LIN {X 0,Y 563.964,Z 599.477,A -85,B 0,C 180,E1 22437.391,E2 22437.391} C_VEL
LIN {X 0,Y 563.324,Z 620.016,A -85,B 0,C 180,E1 22436.115,E2 22436.115} C_VEL
LIN {X 0,Y 562.702,Z 638.754,A -85,B 0,C 180,E1 22434.736,E2 22434.736} C_VEL
LIN {X 0,Y 562.109,Z 656.522,A -85,B 0,C 180,E1 22433.203,E2 22433.203} C_VEL
LIN {X 0,Y 561.587,Z 672.775,A -85,B 0,C 180,E1 22431.57,E2 22431.57} C_VEL
LIN {X 0,Y 561.094,Z 689.022,A -85,B 0,C 180,E1 22429.681,E2 22429.681} C_VEL
LIN {X 0,Y 560.721,Z 703.041,A -85,B 0,C 180,E1 22427.784,E2 22427.784} C_VEL
LIN {X 0,Y 560.419,Z 715.335,A -85,B 0,C 180,E1 22425.841,E2 22425.841} C_VEL
LIN {X 0,Y 560.206,Z 726.094,A -85,B 0,C 180,E1 22423.837,E2 22423.837} C_VEL
LIN {X 0,Y 560.064,Z 735.578,A -85,B 0,C 180,E1 22421.742,E2 22421.742} C_VEL
LIN {X 0,Y 559.974,Z 743.231,A -85,B 0,C 180,E1 22419.662,E2 22419.662} C_VEL
LIN {X 0,Y 559.926,Z 749.535,A -85,B 0,C 180,E1 22417.49,E2 22417.49} C_VEL
LIN {X 0,Y 559.914,Z 754.246,A -85,B 0,C 180,E1 22415.328,E2 22415.328} C_VEL
LIN {X 0,Y 559.914,Z 757.235,A -85,B 0,C 180,E1 22413.173,E2 22413.173} C_VEL
LIN {X 0,Y 559.911,Z 758.795,A -85,B 0,C 180,E1 22410.921,E2 22410.921} C_VEL
LIN {X 0,Y 559.913,Z 758.748,A -85,B 0,C 180,E1 22408.772,E2 22408.772} C_VEL
LIN {X 0,Y 559.916,Z 757.071,A -85,B 0,C 180,E1 22406.586,E2 22406.586} C_VEL
LIN {X 0,Y 559.922,Z 753.812,A -85,B 0,C 180,E1 22404.364,E2 22404.364} C_VEL
LIN {X 0,Y 559.93,Z 749.248,A -85,B 0,C 180,E1 22402.304,E2 22402.304} C_VEL
LIN {X 0,Y 559.978,Z 742.83,A -85,B 0,C 180,E1 22400.13,E2 22400.13} C_VEL
LIN {X 0,Y 560.079,Z 735.084,A -85,B 0,C 180,E1 22398.041,E2 22398.041} C_VEL
LIN {X 0,Y 560.224,Z 725.498,A -85,B 0,C 180,E1 22395.953,E2 22395.953} C_VEL
LIN {X 0,Y 560.45,Z 713.965,A -85,B 0,C 180,E1 22393.841,E2 22393.841} C_VEL
LIN {X 0,Y 560.763,Z 701.306,A -85,B 0,C 180,E1 22391.871,E2 22391.871} C_VEL
LIN {X 0,Y 561.156,Z 687.174,A -85,B 0,C 180,E1 22389.996,E2 22389.996} C_VEL
LIN {X 0,Y 561.628,Z 671.445,A -85,B 0,C 180,E1 22388.197,E2 22388.197} C_VEL
LIN {X 0,Y 562.193,Z 653.882,A -85,B 0,C 180,E1 22386.468,E2 22386.468} C_VEL
LIN {X 0,Y 562.78,Z 636.185,A -85,B 0,C 180,E1 22384.97,E2 22384.97} C_VEL
LIN {X 0,Y 563.41,Z 617.535,A -85,B 0,C 180,E1 22383.626,E2 22383.626} C_VEL
LIN {X 0,Y 564.028,Z 597.68,A -85,B 0,C 180,E1 22382.419,E2 22382.419} C_VEL
LIN {X 0,Y 564.627,Z 577.104,A -85,B 0,C 180,E1 22381.38,E2 22381.38} C_VEL
LIN {X 0,Y 565.175,Z 556.456,A -85,B 0,C 180,E1 22380.541,E2 22380.541} C_VEL
LIN {X 0,Y 565.571,Z 535.019,A -85,B 0,C 180,E1 22379.871,E2 22379.871} C_VEL
LIN {X 0,Y 565.962,Z 512.641,A -85,B 0,C 180,E1 22379.375,E2 22379.375} C_VEL
LIN {X 0,Y 567.326,Z 287.147,A -85,B 0,C 180,E1 22376.127,E2 22376.127} C_VEL
LIN {X 0,Y 567.586,Z 216.731,A -85,B 0,C 180,E1 22375.087,E2 22375.087} C_VEL
LIN {X 0,Y 566.157,Z 208.127,A -85,B 0,C 180,E1 22374.819,E2 22374.819} C_VEL
LIN {X 0,Y 567.277,Z 159.958,A -85,B 0,C 180,E1 22371.59,E2 22371.59} C_VEL
LIN {X 0,Y 567.466,Z 148.971,A -85,B 0,C 180,E1 22370.829,E2 22370.829} C_VEL
LIN {X 0,Y 560.322,Z 132.731,A -85,B 0,C 180,E1 22369.009,E2 22369.009} C_VEL
LIN {X 0,Y 560.266,Z 132.249,A -85,B 0,C 180,E1 22368.542,E2 22368.542} C_VEL
LIN {X 0,Y 560.213,Z 132.266,A -85,B 0,C 180,E1 22365.408,E2 22365.408} C_VEL
LIN {X 0,Y 560.208,Z 132.264,A -85,B 0,C 180,E1 22362.013,E2 22362.013} C_VEL
LIN {X 0,Y 560.234,Z 132.255,A -85,B 0,C 180,E1 22359.051,E2 22359.051} C_VEL
LIN {X 0,Y 560.198,Z 132.249,A -85,B 0,C 180,E1 22355.833,E2 22355.833} C_VEL
LIN {X 0,Y 560.268,Z 132.256,A -85,B 0,C 180,E1 22352.612,E2 22352.612} C_VEL
LIN {X 0,Y 560.213,Z 132.257,A -85,B 0,C 180,E1 22349.431,E2 22349.431} C_VEL
LIN {X 0,Y 560.218,Z 132.25,A -85,B 0,C 180,E1 22346.044,E2 22346.044} C_VEL
LIN {X 0,Y 560.268,Z 132.259,A -85,B 0,C 180,E1 22342.895,E2 22342.895} C_VEL
LIN {X 0,Y 560.215,Z 132.25,A -85,B 0,C 180,E1 22339.714,E2 22339.714} C_VEL
LIN {X 0,Y 560.268,Z 132.258,A -85,B 0,C 180,E1 22336.484,E2 22336.484} C_VEL
LIN {X 0,Y 560.235,Z 132.258,A -85,B 0,C 180,E1 22333.311,E2 22333.311} C_VEL
LIN {X 0,Y 560.23,Z 132.257,A -85,B 0,C 180,E1 22329.969,E2 22329.969} C_VEL
LIN {X 0,Y 560.286,Z 132.258,A -85,B 0,C 180,E1 22326.764,E2 22326.764} C_VEL
LIN {X 0,Y 560.235,Z 132.256,A -85,B 0,C 180,E1 22323.479,E2 22323.479} C_VEL
LIN {X 0,Y 560.244,Z 132.253,A -85,B 0,C 180,E1 22320.102,E2 22320.102} C_VEL
LIN {X 0,Y 560.282,Z 132.256,A -85,B 0,C 180,E1 22316.829,E2 22316.829} C_VEL
LIN {X 0,Y 560.241,Z 132.258,A -85,B 0,C 180,E1 22313.544,E2 22313.544} C_VEL
LIN {X 0,Y 560.263,Z 132.251,A -85,B 0,C 180,E1 22310.239,E2 22310.239} C_VEL
LIN {X 0,Y 560.279,Z 132.254,A -85,B 0,C 180,E1 22306.901,E2 22306.901} C_VEL
LIN {X 0,Y 560.246,Z 132.247,A -85,B 0,C 180,E1 22303.622,E2 22303.622} C_VEL
LIN {X 0,Y 560.274,Z 132.25,A -85,B 0,C 180,E1 22300.288,E2 22300.288} C_VEL
LIN {X 0,Y 560.28,Z 132.252,A -85,B 0,C 180,E1 22296.995,E2 22296.995} C_VEL
LIN {X 0,Y 560.254,Z 132.254,A -85,B 0,C 180,E1 22293.731,E2 22293.731} C_VEL
LIN {X 0,Y 560.283,Z 132.253,A -85,B 0,C 180,E1 22290.375,E2 22290.375} C_VEL
LIN {X 0,Y 560.278,Z 132.249,A -85,B 0,C 180,E1 22287.006,E2 22287.006} C_VEL
LIN {X 0,Y 560.26,Z 132.252,A -85,B 0,C 180,E1 22283.666,E2 22283.666} C_VEL
LIN {X 0,Y 560.28,Z 132.251,A -85,B 0,C 180,E1 22280.292,E2 22280.292} C_VEL
LIN {X 0,Y 560.268,Z 132.254,A -85,B 0,C 180,E1 22276.882,E2 22276.882} C_VEL
LIN {X 0,Y 560.269,Z 132.252,A -85,B 0,C 180,E1 22273.538,E2 22273.538} C_VEL
LIN {X 0,Y 560.346,Z 132.693,A -85,B 0,C 180,E1 22273.213,E2 22273.213} C_VEL
LIN {X 0,Y 561.705,Z 135.907,A -85,B 0,C 180,E1 22272.83,E2 22272.83} C_VEL
LIN {X 0,Y 568.634,Z 150.292,A -85,B 0,C 180,E1 22271.207,E2 22271.207} C_VEL
LIN {X 0,Y 568.491,Z 162.115,A -85,B 0,C 180,E1 22270.464,E2 22270.464} C_VEL
LIN {X 0,Y 570.272,Z 172.641,A -85,B 0,C 180,E1 22270.141,E2 22270.141} C_VEL
LIN {X 0,Y 568.756,Z 379.763,A -85,B 0,C 180,E1 22266.99,E2 22266.99} C_VEL
LIN {X 0,Y 567.81,Z 510.946,A -85,B 0,C 180,E1 22265.019,E2 22265.019} C_VEL
LIN {X 0,Y 567.322,Z 534.795,A -85,B 0,C 180,E1 22264.471,E2 22264.471} C_VEL
LIN {X 0,Y 566.849,Z 556.769,A -85,B 0,C 180,E1 22263.779,E2 22263.779} C_VEL
LIN {X 0,Y 566.165,Z 578.711,A -85,B 0,C 180,E1 22262.891,E2 22262.891} C_VEL
LIN {X 0,Y 565.506,Z 599.807,A -85,B 0,C 180,E1 22261.854,E2 22261.854} C_VEL
LIN {X 0,Y 564.723,Z 620.862,A -85,B 0,C 180,E1 22260.604,E2 22260.604} C_VEL
LIN {X 0,Y 563.958,Z 641.417,A -85,B 0,C 180,E1 22259.179,E2 22259.179} C_VEL
LIN {X 0,Y 563.248,Z 659.599,A -85,B 0,C 180,E1 22257.715,E2 22257.715} C_VEL
LIN {X 0,Y 562.523,Z 678.969,A -85,B 0,C 180,E1 22255.922,E2 22255.922} C_VEL
LIN {X 0,Y 561.905,Z 696.173,A -85,B 0,C 180,E1 22254.1,E2 22254.1} C_VEL
LIN {X 0,Y 561.361,Z 712.099,A -85,B 0,C 180,E1 22252.152,E2 22252.152} C_VEL
LIN {X 0,Y 560.903,Z 727.34,A -85,B 0,C 180,E1 22250.014,E2 22250.014} C_VEL
LIN {X 0,Y 560.562,Z 740.01,A -85,B 0,C 180,E1 22247.973,E2 22247.973} C_VEL
LIN {X 0,Y 560.301,Z 751.321,A -85,B 0,C 180,E1 22245.844,E2 22245.844} C_VEL
LIN {X 0,Y 560.136,Z 761.456,A -85,B 0,C 180,E1 22243.628,E2 22243.628} C_VEL
LIN {X 0,Y 560.026,Z 769.7,A -85,B 0,C 180,E1 22241.429,E2 22241.429} C_VEL
LIN {X 0,Y 559.964,Z 776.775,A -85,B 0,C 180,E1 22239.144,E2 22239.144} C_VEL
LIN {X 0,Y 559.928,Z 782.07,A -85,B 0,C 180,E1 22236.86,E2 22236.86} C_VEL
LIN {X 0,Y 559.899,Z 785.913,A -85,B 0,C 180,E1 22234.609,E2 22234.609} C_VEL
LIN {X 0,Y 559.904,Z 788.122,A -85,B 0,C 180,E1 22232.354,E2 22232.354} C_VEL
LIN {X 0,Y 559.91,Z 788.984,A -85,B 0,C 180,E1 22230.102,E2 22230.102} C_VEL
LIN {X 0,Y 559.905,Z 788.189,A -85,B 0,C 180,E1 22227.749,E2 22227.749} C_VEL
LIN {X 0,Y 559.898,Z 786.049,A -85,B 0,C 180,E1 22225.493,E2 22225.493} C_VEL
LIN {X 0,Y 559.927,Z 782.254,A -85,B 0,C 180,E1 22223.232,E2 22223.232} C_VEL
LIN {X 0,Y 559.952,Z 777.296,A -85,B 0,C 180,E1 22221.063,E2 22221.063} C_VEL
LIN {X 0,Y 560.019,Z 770.409,A -85,B 0,C 180,E1 22218.778,E2 22218.778} C_VEL
LIN {X 0,Y 560.125,Z 762.439,A -85,B 0,C 180,E1 22216.62,E2 22216.62} C_VEL
LIN {X 0,Y 560.282,Z 752.364,A -85,B 0,C 180,E1 22214.368,E2 22214.368} C_VEL
LIN {X 0,Y 560.548,Z 741.242,A -85,B 0,C 180,E1 22212.241,E2 22212.241} C_VEL
LIN {X 0,Y 560.885,Z 728.049,A -85,B 0,C 180,E1 22210.094,E2 22210.094} C_VEL
LIN {X 0,Y 561.317,Z 713.542,A -85,B 0,C 180,E1 22208.034,E2 22208.034} C_VEL
LIN {X 0,Y 561.815,Z 698.473,A -85,B 0,C 180,E1 22206.172,E2 22206.172} C_VEL
LIN {X 0,Y 562.437,Z 681.124,A -85,B 0,C 180,E1 22204.294,E2 22204.294} C_VEL
LIN {X 0,Y 563.12,Z 663.258,A -85,B 0,C 180,E1 22202.596,E2 22202.596} C_VEL
LIN {X 0,Y 563.845,Z 644.352,A -85,B 0,C 180,E1 22201.047,E2 22201.047} C_VEL
LIN {X 0,Y 564.609,Z 623.62,A -85,B 0,C 180,E1 22199.572,E2 22199.572} C_VEL
LIN {X 0,Y 565.353,Z 603.85,A -85,B 0,C 180,E1 22198.375,E2 22198.375} C_VEL
LIN {X 0,Y 566.073,Z 581.179,A -85,B 0,C 180,E1 22197.22,E2 22197.22} C_VEL
LIN {X 0,Y 566.763,Z 559.797,A -85,B 0,C 180,E1 22196.333,E2 22196.333} C_VEL
LIN {X 0,Y 567.282,Z 536.967,A -85,B 0,C 180,E1 22195.59,E2 22195.59} C_VEL
LIN {X 0,Y 567.779,Z 514.194,A -85,B 0,C 180,E1 22195.039,E2 22195.039} C_VEL
LIN {X 0,Y 568.146,Z 469.081,A -85,B 0,C 180,E1 22194.337,E2 22194.337} C_VEL
LIN {X 0,Y 569.615,Z 259.273,A -85,B 0,C 180,E1 22191.19,E2 22191.19} C_VEL
LIN {X 0,Y 570.101,Z 170.611,A -85,B 0,C 180,E1 22189.812,E2 22189.812} C_VEL
LIN {X 0,Y 568.377,Z 161.3,A -85,B 0,C 180,E1 22189.504,E2 22189.504} C_VEL
LIN {X 0,Y 568.463,Z 149.871,A -85,B 0,C 180,E1 22188.749,E2 22188.749} C_VEL
LIN {X 0,Y 561.602,Z 135.762,A -85,B 0,C 180,E1 22187.15,E2 22187.15} C_VEL
LIN {X 0,Y 560.314,Z 132.511,A -85,B 0,C 180,E1 22186.748,E2 22186.748} C_VEL
LIN {X 0,Y 560.271,Z 132.249,A -85,B 0,C 180,E1 22183.539,E2 22183.539} C_VEL
LIN {X 0,Y 560.263,Z 132.252,A -85,B 0,C 180,E1 22180.2,E2 22180.2} C_VEL
LIN {X 0,Y 560.278,Z 132.247,A -85,B 0,C 180,E1 22176.842,E2 22176.842} C_VEL
LIN {X 0,Y 560.275,Z 132.254,A -85,B 0,C 180,E1 22173.465,E2 22173.465} C_VEL
LIN {X 0,Y 560.258,Z 132.257,A -85,B 0,C 180,E1 22170.216,E2 22170.216} C_VEL
LIN {X 0,Y 560.276,Z 132.246,A -85,B 0,C 180,E1 22166.954,E2 22166.954} C_VEL
LIN {X 0,Y 560.282,Z 132.253,A -85,B 0,C 180,E1 22163.562,E2 22163.562} C_VEL
LIN {X 0,Y 560.25,Z 132.254,A -85,B 0,C 180,E1 22160.256,E2 22160.256} C_VEL
LIN {X 0,Y 560.276,Z 132.252,A -85,B 0,C 180,E1 22156.911,E2 22156.911} C_VEL
LIN {X 0,Y 560.283,Z 132.247,A -85,B 0,C 180,E1 22153.519,E2 22153.519} C_VEL
LIN {X 0,Y 560.245,Z 132.254,A -85,B 0,C 180,E1 22150.176,E2 22150.176} C_VEL
LIN {X 0,Y 560.274,Z 132.257,A -85,B 0,C 180,E1 22146.867,E2 22146.867} C_VEL
LIN {X 0,Y 560.278,Z 132.253,A -85,B 0,C 180,E1 22143.478,E2 22143.478} C_VEL
LIN {X 0,Y 560.236,Z 132.255,A -85,B 0,C 180,E1 22140.204,E2 22140.204} C_VEL
LIN {X 0,Y 560.271,Z 132.257,A -85,B 0,C 180,E1 22136.931,E2 22136.931} C_VEL
LIN {X 0,Y 560.263,Z 132.256,A -85,B 0,C 180,E1 22133.647,E2 22133.647} C_VEL
LIN {X 0,Y 560.229,Z 132.258,A -85,B 0,C 180,E1 22130.342,E2 22130.342} C_VEL
LIN {X 0,Y 560.283,Z 132.26,A -85,B 0,C 180,E1 22127.11,E2 22127.11} C_VEL
LIN {X 0,Y 560.232,Z 132.258,A -85,B 0,C 180,E1 22123.941,E2 22123.941} C_VEL
LIN {X 0,Y 560.224,Z 132.25,A -85,B 0,C 180,E1 22120.503,E2 22120.503} C_VEL
LIN {X 0,Y 560.287,Z 132.258,A -85,B 0,C 180,E1 22117.307,E2 22117.307} C_VEL
LIN {X 0,Y 560.217,Z 132.257,A -85,B 0,C 180,E1 22116.289,E2 22116.289} C_VEL
LIN {X 0,Y 559.235,Z 132.381,A -85,B 0,C 180,E1 22115.501,E2 22115.501} C_VEL
LIN {X 0,Y 552.763,Z 133.196,A -85,B 0,C 180,E1 22113.232,E2 22113.232} C_VEL
LIN {X 0,Y 552.295,Z 133.251,A -85,B 0,C 180,E1 22112.713,E2 22112.713} C_VEL
LIN {X 0,Y 552.301,Z 133.241,A -85,B 0,C 180,E1 22109.663,E2 22109.663} C_VEL
LIN {X 0,Y 552.271,Z 133.251,A -85,B 0,C 180,E1 22106.358,E2 22106.358} C_VEL
LIN {X 0,Y 552.33,Z 133.239,A -85,B 0,C 180,E1 22103.141,E2 22103.141} C_VEL
LIN {X 0,Y 552.268,Z 133.241,A -85,B 0,C 180,E1 22099.978,E2 22099.978} C_VEL
LIN {X 0,Y 552.265,Z 133.242,A -85,B 0,C 180,E1 22096.53,E2 22096.53} C_VEL
LIN {X 0,Y 552.324,Z 133.233,A -85,B 0,C 180,E1 22093.303,E2 22093.303} C_VEL
LIN {X 0,Y 552.333,Z 133.515,A -85,B 0,C 180,E1 22091.614,E2 22091.614} C_VEL
LIN {X 0,Y 553.79,Z 136.97,A -85,B 0,C 180,E1 22091.159,E2 22091.159} C_VEL
LIN {X 0,Y 560.859,Z 152.929,A -85,B 0,C 180,E1 22089.346,E2 22089.346} C_VEL
LIN {X 0,Y 559.535,Z 198.989,A -85,B 0,C 180,E1 22086.197,E2 22086.197} C_VEL
LIN {X 0,Y 559.443,Z 209.593,A -85,B 0,C 180,E1 22085.518,E2 22085.518} C_VEL
LIN {X 0,Y 561.184,Z 220.385,A -85,B 0,C 180,E1 22085.223,E2 22085.223} C_VEL
LIN {X 0,Y 559.538,Z 451.649,A -85,B 0,C 180,E1 22081.849,E2 22081.849} C_VEL
LIN {X 0,Y 559.038,Z 516.086,A -85,B 0,C 180,E1 22080.895,E2 22080.895} C_VEL
LIN {X 0,Y 558.577,Z 537.66,A -85,B 0,C 180,E1 22080.38,E2 22080.38} C_VEL
LIN {X 0,Y 558.04,Z 559.572,A -85,B 0,C 180,E1 22079.658,E2 22079.658} C_VEL
LIN {X 0,Y 557.433,Z 580.175,A -85,B 0,C 180,E1 22078.789,E2 22078.789} C_VEL
LIN {X 0,Y 556.7,Z 600.485,A -85,B 0,C 180,E1 22077.721,E2 22077.721} C_VEL
LIN {X 0,Y 555.96,Z 620.409,A -85,B 0,C 180,E1 22076.46,E2 22076.46} C_VEL
LIN {X 0,Y 555.207,Z 639.428,A -85,B 0,C 180,E1 22075.036,E2 22075.036} C_VEL
LIN {X 0,Y 554.523,Z 657.135,A -85,B 0,C 180,E1 22073.483,E2 22073.483} C_VEL
LIN {X 0,Y 553.901,Z 673.288,A -85,B 0,C 180,E1 22071.829,E2 22071.829} C_VEL
LIN {X 0,Y 553.335,Z 689.028,A -85,B 0,C 180,E1 22069.969,E2 22069.969} C_VEL
LIN {X 0,Y 552.899,Z 702.546,A -85,B 0,C 180,E1 22068.122,E2 22068.122} C_VEL
LIN {X 0,Y 552.546,Z 714.702,A -85,B 0,C 180,E1 22066.18,E2 22066.18} C_VEL
LIN {X 0,Y 552.274,Z 726.098,A -85,B 0,C 180,E1 22064.04,E2 22064.04} C_VEL
LIN {X 0,Y 552.101,Z 735.581,A -85,B 0,C 180,E1 22061.914,E2 22061.914} C_VEL
LIN {X 0,Y 551.991,Z 743.233,A -85,B 0,C 180,E1 22059.803,E2 22059.803} C_VEL
LIN {X 0,Y 551.934,Z 749.537,A -85,B 0,C 180,E1 22057.599,E2 22057.599} C_VEL
LIN {X 0,Y 551.917,Z 754.247,A -85,B 0,C 180,E1 22055.405,E2 22055.405} C_VEL
LIN {X 0,Y 551.915,Z 757.236,A -85,B 0,C 180,E1 22053.219,E2 22053.219} C_VEL
LIN {X 0,Y 551.911,Z 758.795,A -85,B 0,C 180,E1 22050.934,E2 22050.934} C_VEL
LIN {X 0,Y 551.912,Z 758.747,A -85,B 0,C 180,E1 22048.754,E2 22048.754} C_VEL
LIN {X 0,Y 551.916,Z 757.099,A -85,B 0,C 180,E1 22046.563,E2 22046.563} C_VEL
LIN {X 0,Y 551.923,Z 754.016,A -85,B 0,C 180,E1 22044.386,E2 22044.386} C_VEL
LIN {X 0,Y 551.936,Z 749.442,A -85,B 0,C 180,E1 22042.272,E2 22042.272} C_VEL
LIN {X 0,Y 552.001,Z 742.828,A -85,B 0,C 180,E1 22039.986,E2 22039.986} C_VEL
LIN {X 0,Y 552.118,Z 735.112,A -85,B 0,C 180,E1 22037.874,E2 22037.874} C_VEL
LIN {X 0,Y 552.298,Z 725.496,A -85,B 0,C 180,E1 22035.747,E2 22035.747} C_VEL
LIN {X 0,Y 552.585,Z 713.55,A -85,B 0,C 180,E1 22033.535,E2 22033.535} C_VEL
LIN {X 0,Y 552.952,Z 700.926,A -85,B 0,C 180,E1 22031.553,E2 22031.553} C_VEL
LIN {X 0,Y 553.408,Z 686.898,A -85,B 0,C 180,E1 22029.668,E2 22029.668} C_VEL
LIN {X 0,Y 553.962,Z 671.578,A -85,B 0,C 180,E1 22027.894,E2 22027.894} C_VEL
LIN {X 0,Y 554.644,Z 653.876,A -85,B 0,C 180,E1 22026.128,E2 22026.128} C_VEL
LIN {X 0,Y 555.355,Z 635.933,A -85,B 0,C 180,E1 22024.593,E2 22024.593} C_VEL
LIN {X 0,Y 556.082,Z 617.232,A -85,B 0,C 180,E1 22023.231,E2 22023.231} C_VEL
LIN {X 0,Y 556.796,Z 598.051,A -85,B 0,C 180,E1 22022.052,E2 22022.052} C_VEL
LIN {X 0,Y 557.476,Z 578.365,A -85,B 0,C 180,E1 22021.037,E2 22021.037} C_VEL
LIN {X 0,Y 558.096,Z 557.916,A -85,B 0,C 180,E1 22020.189,E2 22020.189} C_VEL
LIN {X 0,Y 558.599,Z 535.904,A -85,B 0,C 180,E1 22019.481,E2 22019.481} C_VEL
LIN {X 0,Y 559.057,Z 514.147,A -85,B 0,C 180,E1 22018.982,E2 22018.982} C_VEL
LIN {X 0,Y 560.659,Z 290.34,A -85,B 0,C 180,E1 22015.717,E2 22015.717} C_VEL
LIN {X 0,Y 561.013,Z 218.22,A -85,B 0,C 180,E1 22014.641,E2 22014.641} C_VEL
LIN {X 0,Y 559.33,Z 208.674,A -85,B 0,C 180,E1 22014.356,E2 22014.356} C_VEL
LIN {X 0,Y 560.626,Z 160.862,A -85,B 0,C 180,E1 22011.115,E2 22011.115} C_VEL
LIN {X 0,Y 560.804,Z 152.57,A -85,B 0,C 180,E1 22010.534,E2 22010.534} C_VEL
LIN {X 0,Y 553.59,Z 136.647,A -85,B 0,C 180,E1 22008.708,E2 22008.708} C_VEL
LIN {X 0,Y 552.336,Z 133.514,A -85,B 0,C 180,E1 22008.296,E2 22008.296} C_VEL
LIN {X 0,Y 552.29,Z 133.246,A -85,B 0,C 180,E1 22006.247,E2 22006.247} C_VEL
LIN {X 0,Y 552.289,Z 133.241,A -85,B 0,C 180,E1 22003.15,E2 22003.15} C_VEL
LIN {X 0,Y 552.26,Z 133.242,A -85,B 0,C 180,E1 21999.859,E2 21999.859} C_VEL
LIN {X 0,Y 552.329,Z 133.237,A -85,B 0,C 180,E1 21996.683,E2 21996.683} C_VEL
LIN {X 0,Y 552.27,Z 133.252,A -85,B 0,C 180,E1 21993.426,E2 21993.426} C_VEL
LIN {X 0,Y 552.272,Z 133.245,A -85,B 0,C 180,E1 21989.979,E2 21989.979} C_VEL
LIN {X 0,Y 552.334,Z 133.241,A -85,B 0,C 180,E1 21986.792,E2 21986.792} C_VEL
LIN {X 0,Y 552.274,Z 133.246,A -85,B 0,C 180,E1 21983.585,E2 21983.585} C_VEL
LIN {X 0,Y 552.307,Z 133.236,A -85,B 0,C 180,E1 21980.327,E2 21980.327} C_VEL
LIN {X 0,Y 552.305,Z 133.244,A -85,B 0,C 180,E1 21977.163,E2 21977.163} C_VEL
LIN {X 0,Y 552.284,Z 133.246,A -85,B 0,C 180,E1 21973.826,E2 21973.826} C_VEL
LIN {X 0,Y 552.341,Z 133.245,A -85,B 0,C 180,E1 21970.604,E2 21970.604} C_VEL
LIN {X 0,Y 552.298,Z 133.247,A -85,B 0,C 180,E1 21967.385,E2 21967.385} C_VEL
LIN {X 0,Y 552.296,Z 133.242,A -85,B 0,C 180,E1 21963.945,E2 21963.945} C_VEL
LIN {X 0,Y 552.346,Z 133.241,A -85,B 0,C 180,E1 21960.622,E2 21960.622} C_VEL
LIN {X 0,Y 552.312,Z 133.249,A -85,B 0,C 180,E1 21957.302,E2 21957.302} C_VEL
LIN {X 0,Y 552.305,Z 133.244,A -85,B 0,C 180,E1 21953.973,E2 21953.973} C_VEL
LIN {X 0,Y 552.342,Z 133.243,A -85,B 0,C 180,E1 21950.729,E2 21950.729} C_VEL
LIN {X 0,Y 552.312,Z 133.248,A -85,B 0,C 180,E1 21947.453,E2 21947.453} C_VEL
LIN {X 0,Y 552.312,Z 133.232,A -85,B 0,C 180,E1 21943.997,E2 21943.997} C_VEL
LIN {X 0,Y 552.34,Z 133.241,A -85,B 0,C 180,E1 21940.654,E2 21940.654} C_VEL
LIN {X 0,Y 552.327,Z 133.235,A -85,B 0,C 180,E1 21937.32,E2 21937.32} C_VEL
LIN {X 0,Y 552.317,Z 133.241,A -85,B 0,C 180,E1 21933.881,E2 21933.881} C_VEL
LIN {X 0,Y 552.341,Z 133.244,A -85,B 0,C 180,E1 21930.503,E2 21930.503} C_VEL
LIN {X 0,Y 552.34,Z 133.235,A -85,B 0,C 180,E1 21927.108,E2 21927.108} C_VEL
LIN {X 0,Y 552.321,Z 133.239,A -85,B 0,C 180,E1 21923.704,E2 21923.704} C_VEL
LIN {X 0,Y 552.337,Z 133.241,A -85,B 0,C 180,E1 21920.417,E2 21920.417} C_VEL
LIN {X 0,Y 552.332,Z 133.243,A -85,B 0,C 180,E1 21916.964,E2 21916.964} C_VEL
LIN {X 0,Y 552.367,Z 133.494,A -85,B 0,C 180,E1 21913.961,E2 21913.961} C_VEL
LIN {X 0,Y 553.485,Z 136.496,A -85,B 0,C 180,E1 21913.582,E2 21913.582} C_VEL
LIN {X 0,Y 556.957,Z 143.342,A -85,B 0,C 180,E1 21912.757,E2 21912.757} C_VEL
LIN {X 0,Y 562.132,Z 154.349,A -85,B 0,C 180,E1 21911.511,E2 21911.511} C_VEL
LIN {X 0,Y 562.059,Z 162.118,A -85,B 0,C 180,E1 21911.026,E2 21911.026} C_VEL
LIN {X 0,Y 564.139,Z 174.281,A -85,B 0,C 180,E1 21910.641,E2 21910.641} C_VEL
LIN {X 0,Y 562.353,Z 381.163,A -85,B 0,C 180,E1 21907.461,E2 21907.461} C_VEL
LIN {X 0,Y 561.247,Z 511.159,A -85,B 0,C 180,E1 21905.486,E2 21905.486} C_VEL
LIN {X 0,Y 560.693,Z 534.793,A -85,B 0,C 180,E1 21904.938,E2 21904.938} C_VEL
LIN {X 0,Y 560.119,Z 556.816,A -85,B 0,C 180,E1 21904.239,E2 21904.239} C_VEL
LIN {X 0,Y 559.343,Z 578.709,A -85,B 0,C 180,E1 21903.344,E2 21903.344} C_VEL
LIN {X 0,Y 558.544,Z 599.806,A -85,B 0,C 180,E1 21902.299,E2 21902.299} C_VEL
LIN {X 0,Y 557.681,Z 620.064,A -85,B 0,C 180,E1 21901.087,E2 21901.087} C_VEL
LIN {X 0,Y 556.794,Z 639.945,A -85,B 0,C 180,E1 21899.71,E2 21899.71} C_VEL
LIN {X 0,Y 555.936,Z 658.873,A -85,B 0,C 180,E1 21898.176,E2 21898.176} C_VEL
LIN {X 0,Y 555.059,Z 678.357,A -85,B 0,C 180,E1 21896.361,E2 21896.361} C_VEL
LIN {X 0,Y 554.318,Z 695.679,A -85,B 0,C 180,E1 21894.51,E2 21894.51} C_VEL
LIN {X 0,Y 553.659,Z 711.849,A -85,B 0,C 180,E1 21892.51,E2 21892.51} C_VEL
LIN {X 0,Y 553.098,Z 727.342,A -85,B 0,C 180,E1 21890.309,E2 21890.309} C_VEL
LIN {X 0,Y 552.693,Z 740.008,A -85,B 0,C 180,E1 21888.238,E2 21888.238} C_VEL
LIN {X 0,Y 552.382,Z 751.586,A -85,B 0,C 180,E1 21886.023,E2 21886.023} C_VEL
LIN {X 0,Y 552.182,Z 761.455,A -85,B 0,C 180,E1 21883.828,E2 21883.828} C_VEL
LIN {X 0,Y 552.047,Z 769.952,A -85,B 0,C 180,E1 21881.522,E2 21881.522} C_VEL
LIN {X 0,Y 551.97,Z 777.042,A -85,B 0,C 180,E1 21879.172,E2 21879.172} C_VEL
LIN {X 0,Y 551.931,Z 782.167,A -85,B 0,C 180,E1 21876.911,E2 21876.911} C_VEL
LIN {X 0,Y 551.899,Z 786.049,A -85,B 0,C 180,E1 21874.572,E2 21874.572} C_VEL
LIN {X 0,Y 551.904,Z 788.19,A -85,B 0,C 180,E1 21872.284,E2 21872.284} C_VEL
LIN {X 0,Y 551.911,Z 788.984,A -85,B 0,C 180,E1 21869.896,E2 21869.896} C_VEL
LIN {X 0,Y 551.905,Z 788.122,A -85,B 0,C 180,E1 21867.612,E2 21867.612} C_VEL
LIN {X 0,Y 551.902,Z 785.913,A -85,B 0,C 180,E1 21865.324,E2 21865.324} C_VEL
LIN {X 0,Y 551.932,Z 782.048,A -85,B 0,C 180,E1 21863.029,E2 21863.029} C_VEL
LIN {X 0,Y 551.968,Z 776.775,A -85,B 0,C 180,E1 21860.723,E2 21860.723} C_VEL
LIN {X 0,Y 552.05,Z 769.698,A -85,B 0,C 180,E1 21858.403,E2 21858.403} C_VEL
LIN {X 0,Y 552.188,Z 760.997,A -85,B 0,C 180,E1 21856.065,E2 21856.065} C_VEL
LIN {X 0,Y 552.39,Z 751.324,A -85,B 0,C 180,E1 21853.923,E2 21853.923} C_VEL
LIN {X 0,Y 552.712,Z 739.374,A -85,B 0,C 180,E1 21851.654,E2 21851.654} C_VEL
LIN {X 0,Y 553.12,Z 726.633,A -85,B 0,C 180,E1 21849.582,E2 21849.582} C_VEL
LIN {X 0,Y 553.659,Z 711.849,A -85,B 0,C 180,E1 21847.49,E2 21847.49} C_VEL
LIN {X 0,Y 554.318,Z 695.68,A -85,B 0,C 180,E1 21845.49,E2 21845.49} C_VEL
LIN {X 0,Y 555.059,Z 678.357,A -85,B 0,C 180,E1 21843.639,E2 21843.639} C_VEL
LIN {X 0,Y 555.936,Z 658.871,A -85,B 0,C 180,E1 21841.824,E2 21841.824} C_VEL
LIN {X 0,Y 556.832,Z 639.2,A -85,B 0,C 180,E1 21840.233,E2 21840.233} C_VEL
LIN {X 0,Y 557.721,Z 619.169,A -85,B 0,C 180,E1 21838.856,E2 21838.856} C_VEL
LIN {X 0,Y 558.61,Z 597.581,A -85,B 0,C 180,E1 21837.584,E2 21837.584} C_VEL
LIN {X 0,Y 559.411,Z 577.078,A -85,B 0,C 180,E1 21836.583,E2 21836.583} C_VEL
LIN {X 0,Y 560.164,Z 553.974,A -85,B 0,C 180,E1 21835.662,E2 21835.662} C_VEL
LIN {X 0,Y 560.765,Z 532.841,A -85,B 0,C 180,E1 21835.009,E2 21835.009} C_VEL
LIN {X 0,Y 561.261,Z 509.664,A -85,B 0,C 180,E1 21834.488,E2 21834.488} C_VEL
LIN {X 0,Y 563.061,Z 295.011,A -85,B 0,C 180,E1 21831.226,E2 21831.226} C_VEL
LIN {X 0,Y 563.997,Z 172.439,A -85,B 0,C 180,E1 21829.316,E2 21829.316} C_VEL
LIN {X 0,Y 561.941,Z 161.184,A -85,B 0,C 180,E1 21828.936,E2 21828.936} C_VEL
LIN {X 0,Y 561.981,Z 153.607,A -85,B 0,C 180,E1 21828.424,E2 21828.424} C_VEL
LIN {X 0,Y 553.97,Z 137.188,A -85,B 0,C 180,E1 21826.516,E2 21826.516} C_VEL
LIN {X 0,Y 552.381,Z 133.59,A -85,B 0,C 180,E1 21826.063,E2 21826.063} C_VEL
LIN {X 0,Y 552.325,Z 133.23,A -85,B 0,C 180,E1 21825.204,E2 21825.204} C_VEL
LIN {X 0,Y 552.335,Z 133.243,A -85,B 0,C 180,E1 21821.911,E2 21821.911} C_VEL
LIN {X 0,Y 552.329,Z 133.246,A -85,B 0,C 180,E1 21818.515,E2 21818.515} C_VEL
LIN {X 0,Y 552.333,Z 133.244,A -85,B 0,C 180,E1 21815.146,E2 21815.146} C_VEL
LIN {X 0,Y 552.34,Z 133.232,A -85,B 0,C 180,E1 21811.703,E2 21811.703} C_VEL
LIN {X 0,Y 552.317,Z 133.237,A -85,B 0,C 180,E1 21808.313,E2 21808.313} C_VEL
LIN {X 0,Y 552.341,Z 133.247,A -85,B 0,C 180,E1 21804.92,E2 21804.92} C_VEL
LIN {X 0,Y 552.34,Z 133.227,A -85,B 0,C 180,E1 21801.498,E2 21801.498} C_VEL
LIN {X 0,Y 552.312,Z 133.245,A -85,B 0,C 180,E1 21798.142,E2 21798.142} C_VEL
LIN {X 0,Y 552.331,Z 133.233,A -85,B 0,C 180,E1 21794.788,E2 21794.788} C_VEL
LIN {X 0,Y 552.342,Z 133.244,A -85,B 0,C 180,E1 21791.38,E2 21791.38} C_VEL
LIN {X 0,Y 552.305,Z 133.245,A -85,B 0,C 180,E1 21788.117,E2 21788.117} C_VEL
LIN {X 0,Y 552.324,Z 133.248,A -85,B 0,C 180,E1 21784.777,E2 21784.777} C_VEL
LIN {X 0,Y 552.342,Z 133.244,A -85,B 0,C 180,E1 21781.452,E2 21781.452} C_VEL
LIN {X 0,Y 552.297,Z 133.247,A -85,B 0,C 180,E1 21778.236,E2 21778.236} C_VEL
LIN {X 0,Y 552.329,Z 133.251,A -85,B 0,C 180,E1 21774.911,E2 21774.911} C_VEL
LIN {X 0,Y 552.318,Z 133.243,A -85,B 0,C 180,E1 21771.673,E2 21771.673} C_VEL
LIN {X 0,Y 552.289,Z 133.248,A -85,B 0,C 180,E1 21768.348,E2 21768.348} C_VEL
LIN {X 0,Y 552.343,Z 133.245,A -85,B 0,C 180,E1 21765.105,E2 21765.105} C_VEL
LIN {X 0,Y 552.297,Z 133.241,A -85,B 0,C 180,E1 21761.857,E2 21761.857} C_VEL
LIN {X 0,Y 552.284,Z 133.249,A -85,B 0,C 180,E1 21758.438,E2 21758.438} C_VEL
LIN {X 0,Y 552.34,Z 133.234,A -85,B 0,C 180,E1 21755.281,E2 21755.281} C_VEL
LIN {X 0,Y 552.295,Z 133.251,A -85,B 0,C 180,E1 21752.713,E2 21752.713} C_VEL
LIN {X 0,Y 551.284,Z 133.375,A -85,B 0,C 180,E1 21751.915,E2 21751.915} C_VEL
LIN {X 0,Y 544.86,Z 134.165,A -85,B 0,C 180,E1 21749.612,E2 21749.612} C_VEL
LIN {X 0,Y 544.389,Z 134.221,A -85,B 0,C 180,E1 21749.086,E2 21749.086} C_VEL
LIN {X 0,Y 544.339,Z 134.24,A -85,B 0,C 180,E1 21745.928,E2 21745.928} C_VEL
LIN {X 0,Y 544.333,Z 134.242,A -85,B 0,C 180,E1 21742.514,E2 21742.514} C_VEL
LIN {X 0,Y 544.393,Z 134.222,A -85,B 0,C 180,E1 21739.306,E2 21739.306} C_VEL
LIN {X 0,Y 544.324,Z 134.227,A -85,B 0,C 180,E1 21736.025,E2 21736.025} C_VEL
LIN {X 0,Y 544.327,Z 134.218,A -85,B 0,C 180,E1 21732.558,E2 21732.558} C_VEL
LIN {X 0,Y 544.411,Z 134.788,A -85,B 0,C 180,E1 21732.256,E2 21732.256} C_VEL
LIN {X 0,Y 546.085,Z 138.328,A -85,B 0,C 180,E1 21731.794,E2 21731.794} C_VEL
LIN {X 0,Y 554.192,Z 156.442,A -85,B 0,C 180,E1 21729.656,E2 21729.656} C_VEL
LIN {X 0,Y 552.671,Z 202.665,A -85,B 0,C 180,E1 21726.462,E2 21726.462} C_VEL
LIN {X 0,Y 552.635,Z 209.519,A -85,B 0,C 180,E1 21726.027,E2 21726.027} C_VEL
LIN {X 0,Y 554.639,Z 221.894,A -85,B 0,C 180,E1 21725.679,E2 21725.679} C_VEL
LIN {X 0,Y 552.734,Z 453.354,A -85,B 0,C 180,E1 21722.264,E2 21722.264} C_VEL
LIN {X 0,Y 552.17,Z 516.123,A -85,B 0,C 180,E1 21721.322,E2 21721.322} C_VEL
LIN {X 0,Y 551.641,Z 537.725,A -85,B 0,C 180,E1 21720.802,E2 21720.802} C_VEL
LIN {X 0,Y 551.041,Z 559.38,A -85,B 0,C 180,E1 21720.082,E2 21720.082} C_VEL
LIN {X 0,Y 550.351,Z 578.97,A -85,B 0,C 180,E1 21719.255,E2 21719.255} C_VEL
LIN {X 0,Y 549.579,Z 598.514,A -85,B 0,C 180,E1 21718.23,E2 21718.23} C_VEL
LIN {X 0,Y 548.682,Z 619.219,A -85,B 0,C 180,E1 21716.925,E2 21716.925} C_VEL
LIN {X 0,Y 547.837,Z 638.098,A -85,B 0,C 180,E1 21715.513,E2 21715.513} C_VEL
LIN {X 0,Y 547.023,Z 655.937,A -85,B 0,C 180,E1 21713.939,E2 21713.939} C_VEL
LIN {X 0,Y 546.284,Z 672.281,A -85,B 0,C 180,E1 21712.263,E2 21712.263} C_VEL
LIN {X 0,Y 545.615,Z 688.185,A -85,B 0,C 180,E1 21710.376,E2 21710.376} C_VEL
LIN {X 0,Y 545.111,Z 701.833,A -85,B 0,C 180,E1 21708.5,E2 21708.5} C_VEL
LIN {X 0,Y 544.672,Z 714.705,A -85,B 0,C 180,E1 21706.421,E2 21706.421} C_VEL
LIN {X 0,Y 544.349,Z 726.103,A -85,B 0,C 180,E1 21704.248,E2 21704.248} C_VEL
LIN {X 0,Y 544.142,Z 735.585,A -85,B 0,C 180,E1 21702.091,E2 21702.091} C_VEL
LIN {X 0,Y 544.013,Z 743.235,A -85,B 0,C 180,E1 21699.948,E2 21699.948} C_VEL
LIN {X 0,Y 543.946,Z 749.539,A -85,B 0,C 180,E1 21697.711,E2 21697.711} C_VEL
LIN {X 0,Y 543.92,Z 754.248,A -85,B 0,C 180,E1 21695.485,E2 21695.485} C_VEL
LIN {X 0,Y 543.915,Z 757.237,A -85,B 0,C 180,E1 21693.267,E2 21693.267} C_VEL
LIN {X 0,Y 543.912,Z 758.795,A -85,B 0,C 180,E1 21690.948,E2 21690.948} C_VEL
LIN {X 0,Y 543.912,Z 758.747,A -85,B 0,C 180,E1 21688.736,E2 21688.736} C_VEL
LIN {X 0,Y 543.916,Z 757.109,A -85,B 0,C 180,E1 21686.522,E2 21686.522} C_VEL
LIN {X 0,Y 543.926,Z 754.015,A -85,B 0,C 180,E1 21684.303,E2 21684.303} C_VEL
LIN {X 0,Y 543.946,Z 749.499,A -85,B 0,C 180,E1 21682.182,E2 21682.182} C_VEL
LIN {X 0,Y 544.024,Z 742.826,A -85,B 0,C 180,E1 21679.838,E2 21679.838} C_VEL
LIN {X 0,Y 544.159,Z 735.11,A -85,B 0,C 180,E1 21677.694,E2 21677.694} C_VEL
LIN {X 0,Y 544.373,Z 725.494,A -85,B 0,C 180,E1 21675.535,E2 21675.535} C_VEL
LIN {X 0,Y 544.697,Z 713.956,A -85,B 0,C 180,E1 21673.361,E2 21673.361} C_VEL
LIN {X 0,Y 545.118,Z 701.691,A -85,B 0,C 180,E1 21671.389,E2 21671.389} C_VEL
LIN {X 0,Y 545.64,Z 687.557,A -85,B 0,C 180,E1 21669.453,E2 21669.453} C_VEL
LIN {X 0,Y 546.297,Z 672.079,A -85,B 0,C 180,E1 21667.624,E2 21667.624} C_VEL
LIN {X 0,Y 547.061,Z 655.078,A -85,B 0,C 180,E1 21665.891,E2 21665.891} C_VEL
LIN {X 0,Y 547.892,Z 637.11,A -85,B 0,C 180,E1 21664.316,E2 21664.316} C_VEL
LIN {X 0,Y 548.733,Z 618.031,A -85,B 0,C 180,E1 21662.902,E2 21662.902} C_VEL
LIN {X 0,Y 549.602,Z 598.037,A -85,B 0,C 180,E1 21661.653,E2 21661.653} C_VEL
LIN {X 0,Y 550.373,Z 578.352,A -85,B 0,C 180,E1 21660.627,E2 21660.627} C_VEL
LIN {X 0,Y 551.07,Z 558.561,A -85,B 0,C 180,E1 21659.797,E2 21659.797} C_VEL
LIN {X 0,Y 551.666,Z 536.268,A -85,B 0,C 180,E1 21659.067,E2 21659.067} C_VEL
LIN {X 0,Y 552.19,Z 514.575,A -85,B 0,C 180,E1 21658.561,E2 21658.561} C_VEL
LIN {X 0,Y 554.031,Z 292.198,A -85,B 0,C 180,E1 21655.278,E2 21655.278} C_VEL
LIN {X 0,Y 554.473,Z 219.73,A -85,B 0,C 180,E1 21654.185,E2 21654.185} C_VEL
LIN {X 0,Y 552.53,Z 208.66,A -85,B 0,C 180,E1 21653.849,E2 21653.849} C_VEL
LIN {X 0,Y 554.014,Z 161.675,A -85,B 0,C 180,E1 21650.621,E2 21650.621} C_VEL
LIN {X 0,Y 554.144,Z 156.208,A -85,B 0,C 180,E1 21650.233,E2 21650.233} C_VEL
LIN {X 0,Y 546.264,Z 138.605,A -85,B 0,C 180,E1 21648.155,E2 21648.155} C_VEL
LIN {X 0,Y 544.423,Z 134.798,A -85,B 0,C 180,E1 21647.657,E2 21647.657} C_VEL
LIN {X 0,Y 544.336,Z 134.241,A -85,B 0,C 180,E1 21647.44,E2 21647.44} C_VEL
LIN {X 0,Y 544.33,Z 134.226,A -85,B 0,C 180,E1 21643.974,E2 21643.974} C_VEL
LIN {X 0,Y 544.394,Z 134.222,A -85,B 0,C 180,E1 21640.693,E2 21640.693} C_VEL
LIN {X 0,Y 544.327,Z 134.243,A -85,B 0,C 180,E1 21637.446,E2 21637.446} C_VEL
LIN {X 0,Y 544.334,Z 134.241,A -85,B 0,C 180,E1 21634.066,E2 21634.066} C_VEL
LIN {X 0,Y 544.375,Z 134.223,A -85,B 0,C 180,E1 21630.939,E2 21630.939} C_VEL
LIN {X 0,Y 544.331,Z 134.24,A -85,B 0,C 180,E1 21627.693,E2 21627.693} C_VEL
LIN {X 0,Y 544.372,Z 134.228,A -85,B 0,C 180,E1 21624.41,E2 21624.41} C_VEL
LIN {X 0,Y 544.349,Z 134.239,A -85,B 0,C 180,E1 21621.327,E2 21621.327} C_VEL
LIN {X 0,Y 544.343,Z 134.231,A -85,B 0,C 180,E1 21617.928,E2 21617.928} C_VEL
LIN {X 0,Y 544.408,Z 134.231,A -85,B 0,C 180,E1 21614.682,E2 21614.682} C_VEL
LIN {X 0,Y 544.353,Z 134.238,A -85,B 0,C 180,E1 21611.442,E2 21611.442} C_VEL
LIN {X 0,Y 544.357,Z 134.234,A -85,B 0,C 180,E1 21608.025,E2 21608.025} C_VEL
LIN {X 0,Y 544.405,Z 134.232,A -85,B 0,C 180,E1 21604.741,E2 21604.741} C_VEL
LIN {X 0,Y 544.361,Z 134.238,A -85,B 0,C 180,E1 21601.474,E2 21601.474} C_VEL
LIN {X 0,Y 544.364,Z 134.235,A -85,B 0,C 180,E1 21598,E2 21598} C_VEL
LIN {X 0,Y 544.405,Z 134.234,A -85,B 0,C 180,E1 21594.731,E2 21594.731} C_VEL
LIN {X 0,Y 544.37,Z 134.236,A -85,B 0,C 180,E1 21591.444,E2 21591.444} C_VEL
LIN {X 0,Y 544.374,Z 134.233,A -85,B 0,C 180,E1 21588.021,E2 21588.021} C_VEL
LIN {X 0,Y 544.401,Z 134.215,A -85,B 0,C 180,E1 21584.665,E2 21584.665} C_VEL
LIN {X 0,Y 544.39,Z 134.238,A -85,B 0,C 180,E1 21581.252,E2 21581.252} C_VEL
LIN {X 0,Y 544.374,Z 134.218,A -85,B 0,C 180,E1 21577.882,E2 21577.882} C_VEL
LIN {X 0,Y 544.401,Z 134.228,A -85,B 0,C 180,E1 21574.547,E2 21574.547} C_VEL
LIN {X 0,Y 544.402,Z 134.23,A -85,B 0,C 180,E1 21571.117,E2 21571.117} C_VEL
LIN {X 0,Y 544.38,Z 134.222,A -85,B 0,C 180,E1 21567.816,E2 21567.816} C_VEL
LIN {X 0,Y 544.401,Z 134.228,A -85,B 0,C 180,E1 21564.394,E2 21564.394} C_VEL
LIN {X 0,Y 544.396,Z 134.235,A -85,B 0,C 180,E1 21560.953,E2 21560.953} C_VEL
LIN {X 0,Y 544.389,Z 134.238,A -85,B 0,C 180,E1 21557.588,E2 21557.588} C_VEL
LIN {X 0,Y 544.418,Z 134.441,A -85,B 0,C 180,E1 21554.671,E2 21554.671} C_VEL
LIN {X 0,Y 545.717,Z 137.726,A -85,B 0,C 180,E1 21554.243,E2 21554.243} C_VEL
LIN {X 0,Y 554.398,Z 155.194,A -85,B 0,C 180,E1 21552.163,E2 21552.163} C_VEL
LIN {X 0,Y 555.656,Z 158.072,A -85,B 0,C 180,E1 21551.845,E2 21551.845} C_VEL
LIN {X 0,Y 555.709,Z 162.312,A -85,B 0,C 180,E1 21551.594,E2 21551.594} C_VEL
LIN {X 0,Y 558.049,Z 175.949,A -85,B 0,C 180,E1 21551.152,E2 21551.152} C_VEL
LIN {X 0,Y 555.991,Z 382.435,A -85,B 0,C 180,E1 21547.945,E2 21547.945} C_VEL
LIN {X 0,Y 554.726,Z 511.117,A -85,B 0,C 180,E1 21545.968,E2 21545.968} C_VEL
LIN {X 0,Y 554.107,Z 534.791,A -85,B 0,C 180,E1 21545.415,E2 21545.415} C_VEL
LIN {X 0,Y 553.429,Z 556.754,A -85,B 0,C 180,E1 21544.715,E2 21544.715} C_VEL
LIN {X 0,Y 552.557,Z 578.704,A -85,B 0,C 180,E1 21543.808,E2 21543.808} C_VEL
LIN {X 0,Y 551.624,Z 599.867,A -85,B 0,C 180,E1 21542.751,E2 21542.751} C_VEL
LIN {X 0,Y 550.594,Z 620.958,A -85,B 0,C 180,E1 21541.471,E2 21541.471} C_VEL
LIN {X 0,Y 549.503,Z 641.828,A -85,B 0,C 180,E1 21539.99,E2 21539.99} C_VEL
LIN {X 0,Y 548.553,Z 660.265,A -85,B 0,C 180,E1 21538.465,E2 21538.465} C_VEL
LIN {X 0,Y 547.542,Z 679.465,A -85,B 0,C 180,E1 21536.634,E2 21536.634} C_VEL
LIN {X 0,Y 546.691,Z 696.624,A -85,B 0,C 180,E1 21534.76,E2 21534.76} C_VEL
LIN {X 0,Y 545.969,Z 711.848,A -85,B 0,C 180,E1 21532.845,E2 21532.845} C_VEL
LIN {X 0,Y 545.308,Z 727.344,A -85,B 0,C 180,E1 21530.612,E2 21530.612} C_VEL
LIN {X 0,Y 544.846,Z 740.006,A -85,B 0,C 180,E1 21528.51,E2 21528.51} C_VEL
LIN {X 0,Y 544.468,Z 751.845,A -85,B 0,C 180,E1 21526.208,E2 21526.208} C_VEL
LIN {X 0,Y 544.223,Z 761.885,A -85,B 0,C 180,E1 21523.926,E2 21523.926} C_VEL
LIN {X 0,Y 544.069,Z 770.205,A -85,B 0,C 180,E1 21521.618,E2 21521.618} C_VEL
LIN {X 0,Y 543.976,Z 777.297,A -85,B 0,C 180,E1 21519.201,E2 21519.201} C_VEL
LIN {X 0,Y 543.934,Z 782.263,A -85,B 0,C 180,E1 21516.964,E2 21516.964} C_VEL
LIN {X 0,Y 543.901,Z 786.049,A -85,B 0,C 180,E1 21514.639,E2 21514.639} C_VEL
LIN {X 0,Y 543.904,Z 788.19,A -85,B 0,C 180,E1 21512.318,E2 21512.318} C_VEL
LIN {X 0,Y 543.91,Z 788.984,A -85,B 0,C 180,E1 21509.895,E2 21509.895} C_VEL
LIN {X 0,Y 543.906,Z 788.123,A -85,B 0,C 180,E1 21507.577,E2 21507.577} C_VEL
LIN {X 0,Y 543.905,Z 785.913,A -85,B 0,C 180,E1 21505.255,E2 21505.255} C_VEL
LIN {X 0,Y 543.936,Z 782.048,A -85,B 0,C 180,E1 21502.926,E2 21502.926} C_VEL
LIN {X 0,Y 543.973,Z 776.775,A -85,B 0,C 180,E1 21500.585,E2 21500.585} C_VEL
LIN {X 0,Y 544.074,Z 769.699,A -85,B 0,C 180,E1 21498.23,E2 21498.23} C_VEL
LIN {X 0,Y 544.244,Z 760.996,A -85,B 0,C 180,E1 21495.858,E2 21495.858} C_VEL
LIN {X 0,Y 544.486,Z 751.326,A -85,B 0,C 180,E1 21493.683,E2 21493.683} C_VEL
LIN {X 0,Y 544.871,Z 739.372,A -85,B 0,C 180,E1 21491.38,E2 21491.38} C_VEL
LIN {X 0,Y 545.337,Z 726.635,A -85,B 0,C 180,E1 21489.277,E2 21489.277} C_VEL
LIN {X 0,Y 545.99,Z 711.368,A -85,B 0,C 180,E1 21487.092,E2 21487.092} C_VEL
LIN {X 0,Y 546.76,Z 695.418,A -85,B 0,C 180,E1 21485.098,E2 21485.098} C_VEL
LIN {X 0,Y 547.606,Z 678.177,A -85,B 0,C 180,E1 21483.233,E2 21483.233} C_VEL
LIN {X 0,Y 548.621,Z 658.867,A -85,B 0,C 180,E1 21481.413,E2 21481.413} C_VEL
LIN {X 0,Y 549.667,Z 639.198,A -85,B 0,C 180,E1 21479.805,E2 21479.805} C_VEL
LIN {X 0,Y 550.686,Z 619.075,A -85,B 0,C 180,E1 21478.406,E2 21478.406} C_VEL
LIN {X 0,Y 551.717,Z 597.585,A -85,B 0,C 180,E1 21477.128,E2 21477.128} C_VEL
LIN {X 0,Y 552.614,Z 577.421,A -85,B 0,C 180,E1 21476.134,E2 21476.134} C_VEL
LIN {X 0,Y 553.472,Z 554.516,A -85,B 0,C 180,E1 21475.207,E2 21475.207} C_VEL
LIN {X 0,Y 554.163,Z 533.36,A -85,B 0,C 180,E1 21474.546,E2 21474.546} C_VEL
LIN {X 0,Y 554.738,Z 510.093,A -85,B 0,C 180,E1 21474.014,E2 21474.014} C_VEL
LIN {X 0,Y 556.793,Z 297.952,A -85,B 0,C 180,E1 21470.754,E2 21470.754} C_VEL
LIN {X 0,Y 557.913,Z 174.14,A -85,B 0,C 180,E1 21468.805,E2 21468.805} C_VEL
LIN {X 0,Y 555.567,Z 161.3,A -85,B 0,C 180,E1 21468.366,E2 21468.366} C_VEL
LIN {X 0,Y 555.5,Z 157.573,A -85,B 0,C 180,E1 21468.106,E2 21468.106} C_VEL
LIN {X 0,Y 547.878,Z 142.037,A -85,B 0,C 180,E1 21466.276,E2 21466.276} C_VEL
LIN {X 0,Y 544.483,Z 134.795,A -85,B 0,C 180,E1 21465.404,E2 21465.404} C_VEL
LIN {X 0,Y 544.388,Z 134.224,A -85,B 0,C 180,E1 21465.149,E2 21465.149} C_VEL
LIN {X 0,Y 544.4,Z 134.229,A -85,B 0,C 180,E1 21461.785,E2 21461.785} C_VEL
LIN {X 0,Y 544.386,Z 134.233,A -85,B 0,C 180,E1 21458.35,E2 21458.35} C_VEL
LIN {X 0,Y 544.399,Z 134.235,A -85,B 0,C 180,E1 21454.961,E2 21454.961} C_VEL
LIN {X 0,Y 544.401,Z 134.221,A -85,B 0,C 180,E1 21451.552,E2 21451.552} C_VEL
LIN {X 0,Y 544.378,Z 134.225,A -85,B 0,C 180,E1 21448.285,E2 21448.285} C_VEL
LIN {X 0,Y 544.4,Z 134.237,A -85,B 0,C 180,E1 21444.87,E2 21444.87} C_VEL
LIN {X 0,Y 544.401,Z 134.214,A -85,B 0,C 180,E1 21441.437,E2 21441.437} C_VEL
LIN {X 0,Y 544.375,Z 134.234,A -85,B 0,C 180,E1 21438.083,E2 21438.083} C_VEL
LIN {X 0,Y 544.384,Z 134.221,A -85,B 0,C 180,E1 21434.682,E2 21434.682} C_VEL
LIN {X 0,Y 544.403,Z 134.233,A -85,B 0,C 180,E1 21431.333,E2 21431.333} C_VEL
LIN {X 0,Y 544.37,Z 134.233,A -85,B 0,C 180,E1 21428.024,E2 21428.024} C_VEL
LIN {X 0,Y 544.375,Z 134.236,A -85,B 0,C 180,E1 21424.635,E2 21424.635} C_VEL
LIN {X 0,Y 544.406,Z 134.235,A -85,B 0,C 180,E1 21421.263,E2 21421.263} C_VEL
LIN {X 0,Y 544.364,Z 134.235,A -85,B 0,C 180,E1 21418,E2 21418} C_VEL
LIN {X 0,Y 544.361,Z 134.238,A -85,B 0,C 180,E1 21414.519,E2 21414.519} C_VEL
LIN {X 0,Y 544.406,Z 134.234,A -85,B 0,C 180,E1 21411.232,E2 21411.232} C_VEL
LIN {X 0,Y 544.359,Z 134.235,A -85,B 0,C 180,E1 21407.913,E2 21407.913} C_VEL
LIN {X 0,Y 544.355,Z 134.239,A -85,B 0,C 180,E1 21404.554,E2 21404.554} C_VEL
LIN {X 0,Y 544.403,Z 134.218,A -85,B 0,C 180,E1 21401.252,E2 21401.252} C_VEL
LIN {X 0,Y 544.346,Z 134.237,A -85,B 0,C 180,E1 21397.994,E2 21397.994} C_VEL
LIN {X 0,Y 544.344,Z 134.223,A -85,B 0,C 180,E1 21394.544,E2 21394.544} C_VEL
LIN {X 0,Y 544.404,Z 134.236,A -85,B 0,C 180,E1 21391.237,E2 21391.237} C_VEL
LIN {X 0,Y 544.389,Z 134.221,A -85,B 0,C 180,E1 21389.086,E2 21389.086} C_VEL
LIN {X 0,Y 543.331,Z 134.358,A -85,B 0,C 180,E1 21388.276,E2 21388.276} C_VEL
LIN {X 0,Y 536.923,Z 135.169,A -85,B 0,C 180,E1 21386,E2 21386} C_VEL
LIN {X 0,Y 536.447,Z 135.218,A -85,B 0,C 180,E1 21385.407,E2 21385.407} C_VEL
LIN {X 0,Y 536.388,Z 135.231,A -85,B 0,C 180,E1 21382.173,E2 21382.173} C_VEL
LIN {X 0,Y 536.429,Z 135.216,A -85,B 0,C 180,E1 21378.997,E2 21378.997} C_VEL
LIN {X 0,Y 536.397,Z 135.212,A -85,B 0,C 180,E1 21375.801,E2 21375.801} C_VEL
LIN {X 0,Y 536.461,Z 135.403,A -85,B 0,C 180,E1 21373.062,E2 21373.062} C_VEL
LIN {X 0,Y 537.325,Z 138.071,A -85,B 0,C 180,E1 21372.691,E2 21372.691} C_VEL
LIN {X 0,Y 542.07,Z 147.534,A -85,B 0,C 180,E1 21371.465,E2 21371.465} C_VEL
LIN {X 0,Y 547.595,Z 160.134,A -85,B 0,C 180,E1 21369.972,E2 21369.972} C_VEL
LIN {X 0,Y 545.818,Z 206.341,A -85,B 0,C 180,E1 21366.733,E2 21366.733} C_VEL
LIN {X 0,Y 545.955,Z 210.039,A -85,B 0,C 180,E1 21366.527,E2 21366.527} C_VEL
LIN {X 0,Y 548.13,Z 223.427,A -85,B 0,C 180,E1 21366.146,E2 21366.146} C_VEL
LIN {X 0,Y 545.955,Z 455.313,A -85,B 0,C 180,E1 21362.685,E2 21362.685} C_VEL
LIN {X 0,Y 545.334,Z 516.158,A -85,B 0,C 180,E1 21361.76,E2 21361.76} C_VEL
LIN {X 0,Y 544.736,Z 537.8,A -85,B 0,C 180,E1 21361.235,E2 21361.235} C_VEL
LIN {X 0,Y 544.065,Z 559.396,A -85,B 0,C 180,E1 21360.508,E2 21360.508} C_VEL
LIN {X 0,Y 543.279,Z 578.989,A -85,B 0,C 180,E1 21359.673,E2 21359.673} C_VEL
LIN {X 0,Y 542.41,Z 598.523,A -85,B 0,C 180,E1 21358.637,E2 21358.637} C_VEL
LIN {X 0,Y 541.396,Z 618.958,A -85,B 0,C 180,E1 21357.337,E2 21357.337} C_VEL
LIN {X 0,Y 540.494,Z 637.165,A -85,B 0,C 180,E1 21355.966,E2 21355.966} C_VEL
LIN {X 0,Y 539.526,Z 655.41,A -85,B 0,C 180,E1 21354.345,E2 21354.345} C_VEL
LIN {X 0,Y 538.653,Z 672.287,A -85,B 0,C 180,E1 21352.596,E2 21352.596} C_VEL
LIN {X 0,Y 537.884,Z 688.191,A -85,B 0,C 180,E1 21350.682,E2 21350.682} C_VEL
LIN {X 0,Y 537.283,Z 702.372,A -85,B 0,C 180,E1 21348.697,E2 21348.697} C_VEL
LIN {X 0,Y 536.803,Z 714.707,A -85,B 0,C 180,E1 21346.669,E2 21346.669} C_VEL
LIN {X 0,Y 536.428,Z 726.107,A -85,B 0,C 180,E1 21344.463,E2 21344.463} C_VEL
LIN {X 0,Y 536.185,Z 735.588,A -85,B 0,C 180,E1 21342.273,E2 21342.273} C_VEL
LIN {X 0,Y 536.039,Z 743.237,A -85,B 0,C 180,E1 21340.098,E2 21340.098} C_VEL
LIN {X 0,Y 535.961,Z 749.54,A -85,B 0,C 180,E1 21337.827,E2 21337.827} C_VEL
LIN {X 0,Y 535.924,Z 754.249,A -85,B 0,C 180,E1 21335.567,E2 21335.567} C_VEL
LIN {X 0,Y 535.915,Z 757.238,A -85,B 0,C 180,E1 21333.316,E2 21333.316} C_VEL
LIN {X 0,Y 535.912,Z 758.794,A -85,B 0,C 180,E1 21330.962,E2 21330.962} C_VEL
LIN {X 0,Y 535.911,Z 758.747,A -85,B 0,C 180,E1 21328.717,E2 21328.717} C_VEL
LIN {X 0,Y 535.914,Z 757.109,A -85,B 0,C 180,E1 21326.47,E2 21326.47} C_VEL
LIN {X 0,Y 535.929,Z 754.014,A -85,B 0,C 180,E1 21324.218,E2 21324.218} C_VEL
LIN {X 0,Y 535.96,Z 749.497,A -85,B 0,C 180,E1 21322.065,E2 21322.065} C_VEL
LIN {X 0,Y 536.045,Z 742.823,A -85,B 0,C 180,E1 21319.685,E2 21319.685} C_VEL
LIN {X 0,Y 536.2,Z 735.108,A -85,B 0,C 180,E1 21317.508,E2 21317.508} C_VEL
LIN {X 0,Y 536.446,Z 725.492,A -85,B 0,C 180,E1 21315.317,E2 21315.317} C_VEL
LIN {X 0,Y 536.824,Z 713.951,A -85,B 0,C 180,E1 21313.109,E2 21313.109} C_VEL
LIN {X 0,Y 537.317,Z 701.685,A -85,B 0,C 180,E1 21311.109,E2 21311.109} C_VEL
LIN {X 0,Y 537.893,Z 688.01,A -85,B 0,C 180,E1 21309.205,E2 21309.205} C_VEL
LIN {X 0,Y 538.663,Z 672.071,A -85,B 0,C 180,E1 21307.289,E2 21307.289} C_VEL
LIN {X 0,Y 539.545,Z 655.012,A -85,B 0,C 180,E1 21305.527,E2 21305.527} C_VEL
LIN {X 0,Y 540.496,Z 637.102,A -85,B 0,C 180,E1 21303.938,E2 21303.938} C_VEL
LIN {X 0,Y 541.447,Z 618.018,A -85,B 0,C 180,E1 21302.507,E2 21302.507} C_VEL
LIN {X 0,Y 542.435,Z 598.021,A -85,B 0,C 180,E1 21301.244,E2 21301.244} C_VEL
LIN {X 0,Y 543.312,Z 578.34,A -85,B 0,C 180,E1 21300.207,E2 21300.207} C_VEL
LIN {X 0,Y 544.097,Z 558.539,A -85,B 0,C 180,E1 21299.368,E2 21299.368} C_VEL
LIN {X 0,Y 544.777,Z 536.24,A -85,B 0,C 180,E1 21298.632,E2 21298.632} C_VEL
LIN {X 0,Y 545.356,Z 514.618,A -85,B 0,C 180,E1 21298.122,E2 21298.122} C_VEL
LIN {X 0,Y 547.439,Z 293.802,A -85,B 0,C 180,E1 21294.825,E2 21294.825} C_VEL
LIN {X 0,Y 547.951,Z 221.129,A -85,B 0,C 180,E1 21293.714,E2 21293.714} C_VEL
LIN {X 0,Y 545.773,Z 208.646,A -85,B 0,C 180,E1 21293.329,E2 21293.329} C_VEL
LIN {X 0,Y 547.479,Z 162.851,A -85,B 0,C 180,E1 21290.133,E2 21290.133} C_VEL
LIN {X 0,Y 547.538,Z 159.962,A -85,B 0,C 180,E1 21289.919,E2 21289.919} C_VEL
LIN {X 0,Y 540.074,Z 143.369,A -85,B 0,C 180,E1 21287.92,E2 21287.92} C_VEL
LIN {X 0,Y 536.525,Z 135.755,A -85,B 0,C 180,E1 21286.931,E2 21286.931} C_VEL
LIN {X 0,Y 536.45,Z 135.205,A -85,B 0,C 180,E1 21286.627,E2 21286.627} C_VEL
LIN {X 0,Y 536.394,Z 135.216,A -85,B 0,C 180,E1 21283.368,E2 21283.368} C_VEL
LIN {X 0,Y 536.387,Z 135.215,A -85,B 0,C 180,E1 21279.994,E2 21279.994} C_VEL
LIN {X 0,Y 536.448,Z 135.212,A -85,B 0,C 180,E1 21276.733,E2 21276.733} C_VEL
LIN {X 0,Y 536.391,Z 135.23,A -85,B 0,C 180,E1 21273.488,E2 21273.488} C_VEL
LIN {X 0,Y 536.4,Z 135.22,A -85,B 0,C 180,E1 21270.094,E2 21270.094} C_VEL
LIN {X 0,Y 536.44,Z 135.221,A -85,B 0,C 180,E1 21266.931,E2 21266.931} C_VEL
LIN {X 0,Y 536.397,Z 135.223,A -85,B 0,C 180,E1 21263.626,E2 21263.626} C_VEL
LIN {X 0,Y 536.425,Z 135.211,A -85,B 0,C 180,E1 21260.285,E2 21260.285} C_VEL
LIN {X 0,Y 536.441,Z 135.221,A -85,B 0,C 180,E1 21257.016,E2 21257.016} C_VEL
LIN {X 0,Y 536.405,Z 135.223,A -85,B 0,C 180,E1 21253.694,E2 21253.694} C_VEL
LIN {X 0,Y 536.446,Z 135.223,A -85,B 0,C 180,E1 21250.416,E2 21250.416} C_VEL
LIN {X 0,Y 536.434,Z 135.223,A -85,B 0,C 180,E1 21247.174,E2 21247.174} C_VEL
LIN {X 0,Y 536.416,Z 135.22,A -85,B 0,C 180,E1 21243.848,E2 21243.848} C_VEL
LIN {X 0,Y 536.467,Z 135.217,A -85,B 0,C 180,E1 21240.534,E2 21240.534} C_VEL
LIN {X 0,Y 536.449,Z 135.224,A -85,B 0,C 180,E1 21237.116,E2 21237.116} C_VEL
LIN {X 0,Y 536.423,Z 135.223,A -85,B 0,C 180,E1 21233.794,E2 21233.794} C_VEL
LIN {X 0,Y 536.461,Z 135.217,A -85,B 0,C 180,E1 21230.452,E2 21230.452} C_VEL
LIN {X 0,Y 536.46,Z 135.222,A -85,B 0,C 180,E1 21227.076,E2 21227.076} C_VEL
LIN {X 0,Y 536.43,Z 135.208,A -85,B 0,C 180,E1 21223.717,E2 21223.717} C_VEL
LIN {X 0,Y 536.456,Z 135.216,A -85,B 0,C 180,E1 21220.285,E2 21220.285} C_VEL
LIN {X 0,Y 536.46,Z 135.218,A -85,B 0,C 180,E1 21216.842,E2 21216.842} C_VEL
LIN {X 0,Y 536.446,Z 135.212,A -85,B 0,C 180,E1 21213.428,E2 21213.428} C_VEL
LIN {X 0,Y 536.448,Z 135.223,A -85,B 0,C 180,E1 21210.032,E2 21210.032} C_VEL
LIN {X 0,Y 536.457,Z 135.216,A -85,B 0,C 180,E1 21206.612,E2 21206.612} C_VEL
LIN {X 0,Y 536.459,Z 135.207,A -85,B 0,C 180,E1 21203.253,E2 21203.253} C_VEL
LIN {X 0,Y 536.447,Z 135.212,A -85,B 0,C 180,E1 21199.832,E2 21199.832} C_VEL
LIN {X 0,Y 536.455,Z 135.207,A -85,B 0,C 180,E1 21196.469,E2 21196.469} C_VEL
LIN {X 0,Y 536.49,Z 135.456,A -85,B 0,C 180,E1 21195.391,E2 21195.391} C_VEL
LIN {X 0,Y 537.987,Z 139.016,A -85,B 0,C 180,E1 21194.92,E2 21194.92} C_VEL
LIN {X 0,Y 548.559,Z 160.41,A -85,B 0,C 180,E1 21192.345,E2 21192.345} C_VEL
LIN {X 0,Y 549.416,Z 162.509,A -85,B 0,C 180,E1 21192.176,E2 21192.176} C_VEL
LIN {X 0,Y 552.004,Z 177.717,A -85,B 0,C 180,E1 21191.673,E2 21191.673} C_VEL
LIN {X 0,Y 549.662,Z 384.344,A -85,B 0,C 180,E1 21188.43,E2 21188.43} C_VEL
LIN {X 0,Y 548.243,Z 511.315,A -85,B 0,C 180,E1 21186.458,E2 21186.458} C_VEL
LIN {X 0,Y 547.56,Z 534.789,A -85,B 0,C 180,E1 21185.904,E2 21185.904} C_VEL
LIN {X 0,Y 546.779,Z 556.639,A -85,B 0,C 180,E1 21185.203,E2 21185.203} C_VEL
LIN {X 0,Y 545.817,Z 578.492,A -85,B 0,C 180,E1 21184.293,E2 21184.293} C_VEL
LIN {X 0,Y 544.809,Z 598.704,A -85,B 0,C 180,E1 21183.279,E2 21183.279} C_VEL
LIN {X 0,Y 543.656,Z 619.48,A -85,B 0,C 180,E1 21182.023,E2 21182.023} C_VEL
LIN {X 0,Y 542.485,Z 639.939,A -85,B 0,C 180,E1 21180.576,E2 21180.576} C_VEL
LIN {X 0,Y 541.331,Z 658.943,A -85,B 0,C 180,E1 21179.002,E2 21179.002} C_VEL
LIN {X 0,Y 540.179,Z 678.159,A -85,B 0,C 180,E1 21177.167,E2 21177.167} C_VEL
LIN {X 0,Y 539.217,Z 695.275,A -85,B 0,C 180,E1 21175.291,E2 21175.291} C_VEL
LIN {X 0,Y 538.345,Z 711.001,A -85,B 0,C 180,E1 21173.303,E2 21173.303} C_VEL
LIN {X 0,Y 537.609,Z 725.928,A -85,B 0,C 180,E1 21171.149,E2 21171.149} C_VEL
LIN {X 0,Y 537.058,Z 738.734,A -85,B 0,C 180,E1 21169.014,E2 21169.014} C_VEL
LIN {X 0,Y 536.607,Z 750.804,A -85,B 0,C 180,E1 21166.675,E2 21166.675} C_VEL
LIN {X 0,Y 536.315,Z 760.535,A -85,B 0,C 180,E1 21164.466,E2 21164.466} C_VEL
LIN {X 0,Y 536.107,Z 769.344,A -85,B 0,C 180,E1 21162.057,E2 21162.057} C_VEL
LIN {X 0,Y 535.991,Z 775.869,A -85,B 0,C 180,E1 21159.882,E2 21159.882} C_VEL
LIN {X 0,Y 535.939,Z 781.635,A -85,B 0,C 180,E1 21157.396,E2 21157.396} C_VEL
LIN {X 0,Y 535.916,Z 785.277,A -85,B 0,C 180,E1 21155.245,E2 21155.245} C_VEL
LIN {X 0,Y 535.916,Z 787.988,A -85,B 0,C 180,E1 21152.673,E2 21152.673} C_VEL
LIN {X 0,Y 535.898,Z 788.917,A -85,B 0,C 180,E1 21150.428,E2 21150.428} C_VEL
LIN {X 0,Y 535.909,Z 788.391,A -85,B 0,C 180,E1 21147.969,E2 21147.969} C_VEL
LIN {X 0,Y 535.908,Z 786.617,A -85,B 0,C 180,E1 21145.827,E2 21145.827} C_VEL
LIN {X 0,Y 535.934,Z 783.081,A -85,B 0,C 180,E1 21143.358,E2 21143.358} C_VEL
LIN {X 0,Y 535.958,Z 778.573,A -85,B 0,C 180,E1 21141.201,E2 21141.201} C_VEL
LIN {X 0,Y 536.064,Z 772.178,A -85,B 0,C 180,E1 21138.815,E2 21138.815} C_VEL
LIN {X 0,Y 536.218,Z 764.341,A -85,B 0,C 180,E1 21136.522,E2 21136.522} C_VEL
LIN {X 0,Y 536.47,Z 754.944,A -85,B 0,C 180,E1 21134.211,E2 21134.211} C_VEL
LIN {X 0,Y 536.842,Z 744.15,A -85,B 0,C 180,E1 21131.991,E2 21131.991} C_VEL
LIN {X 0,Y 537.393,Z 730.868,A -85,B 0,C 180,E1 21129.64,E2 21129.64} C_VEL
LIN {X 0,Y 538.014,Z 717.566,A -85,B 0,C 180,E1 21127.606,E2 21127.606} C_VEL
LIN {X 0,Y 538.862,Z 701.273,A -85,B 0,C 180,E1 21125.442,E2 21125.442} C_VEL
LIN {X 0,Y 539.841,Z 684.443,A -85,B 0,C 180,E1 21123.49,E2 21123.49} C_VEL
LIN {X 0,Y 540.865,Z 666.585,A -85,B 0,C 180,E1 21121.695,E2 21121.695} C_VEL
LIN {X 0,Y 542.071,Z 646.54,A -85,B 0,C 180,E1 21119.949,E2 21119.949} C_VEL
LIN {X 0,Y 543.279,Z 626.489,A -85,B 0,C 180,E1 21118.442,E2 21118.442} C_VEL
LIN {X 0,Y 544.415,Z 605.85,A -85,B 0,C 180,E1 21117.133,E2 21117.133} C_VEL
LIN {X 0,Y 545.495,Z 585.082,A -85,B 0,C 180,E1 21116.011,E2 21116.011} C_VEL
LIN {X 0,Y 546.46,Z 564.227,A -85,B 0,C 180,E1 21115.095,E2 21115.095} C_VEL
LIN {X 0,Y 547.343,Z 542.2,A -85,B 0,C 180,E1 21114.31,E2 21114.31} C_VEL
LIN {X 0,Y 547.982,Z 519.893,A -85,B 0,C 180,E1 21113.72,E2 21113.72} C_VEL
LIN {X 0,Y 548.529,Z 492.111,A -85,B 0,C 180,E1 21113.222,E2 21113.222} C_VEL
LIN {X 0,Y 550.806,Z 280.725,A -85,B 0,C 180,E1 21109.957,E2 21109.957} C_VEL
LIN {X 0,Y 551.872,Z 175.855,A -85,B 0,C 180,E1 21108.283,E2 21108.283} C_VEL
LIN {X 0,Y 549.078,Z 161.523,A -85,B 0,C 180,E1 21107.77,E2 21107.77} C_VEL
LIN {X 0,Y 539.991,Z 143.066,A -85,B 0,C 180,E1 21105.582,E2 21105.582} C_VEL
LIN {X 0,Y 536.532,Z 135.68,A -85,B 0,C 180,E1 21104.658,E2 21104.658} C_VEL
LIN {X 0,Y 536.447,Z 135.198,A -85,B 0,C 180,E1 21104.3,E2 21104.3} C_VEL
LIN {X 0,Y 536.462,Z 135.206,A -85,B 0,C 180,E1 21100.858,E2 21100.858} C_VEL
LIN {X 0,Y 536.455,Z 135.211,A -85,B 0,C 180,E1 21097.416,E2 21097.416} C_VEL
LIN {X 0,Y 536.449,Z 135.221,A -85,B 0,C 180,E1 21093.997,E2 21093.997} C_VEL
LIN {X 0,Y 536.45,Z 135.226,A -85,B 0,C 180,E1 21090.563,E2 21090.563} C_VEL
LIN {X 0,Y 536.456,Z 135.205,A -85,B 0,C 180,E1 21087.17,E2 21087.17} C_VEL
LIN {X 0,Y 536.459,Z 135.22,A -85,B 0,C 180,E1 21083.74,E2 21083.74} C_VEL
LIN {X 0,Y 536.435,Z 135.22,A -85,B 0,C 180,E1 21080.284,E2 21080.284} C_VEL
LIN {X 0,Y 536.458,Z 135.214,A -85,B 0,C 180,E1 21076.903,E2 21076.903} C_VEL
LIN {X 0,Y 536.465,Z 135.212,A -85,B 0,C 180,E1 21073.472,E2 21073.472} C_VEL
LIN {X 0,Y 536.431,Z 135.219,A -85,B 0,C 180,E1 21070.091,E2 21070.091} C_VEL
LIN {X 0,Y 536.438,Z 135.224,A -85,B 0,C 180,E1 21066.636,E2 21066.636} C_VEL
LIN {X 0,Y 536.464,Z 135.22,A -85,B 0,C 180,E1 21063.312,E2 21063.312} C_VEL
LIN {X 0,Y 536.427,Z 135.219,A -85,B 0,C 180,E1 21060,E2 21060} C_VEL
LIN {X 0,Y 536.426,Z 135.221,A -85,B 0,C 180,E1 21056.58,E2 21056.58} C_VEL
LIN {X 0,Y 536.468,Z 135.223,A -85,B 0,C 180,E1 21053.257,E2 21053.257} C_VEL
LIN {X 0,Y 536.423,Z 135.224,A -85,B 0,C 180,E1 21049.909,E2 21049.909} C_VEL
LIN {X 0,Y 536.417,Z 135.224,A -85,B 0,C 180,E1 21046.526,E2 21046.526} C_VEL
LIN {X 0,Y 536.465,Z 135.224,A -85,B 0,C 180,E1 21043.208,E2 21043.208} C_VEL
LIN {X 0,Y 536.411,Z 135.211,A -85,B 0,C 180,E1 21039.942,E2 21039.942} C_VEL
LIN {X 0,Y 536.406,Z 135.223,A -85,B 0,C 180,E1 21036.491,E2 21036.491} C_VEL
LIN {X 0,Y 536.459,Z 135.214,A -85,B 0,C 180,E1 21033.189,E2 21033.189} C_VEL
LIN {X 0,Y 536.4,Z 135.221,A -85,B 0,C 180,E1 21030.029,E2 21030.029} C_VEL
LIN {X 0,Y 536.398,Z 135.23,A -85,B 0,C 180,E1 21026.513,E2 21026.513} C_VEL
LIN {X 0,Y 536.447,Z 135.218,A -85,B 0,C 180,E1 21025.407,E2 21025.407} C_VEL
LIN {X 0,Y 535.621,Z 135.309,A -85,B 0,C 180,E1 21024.642,E2 21024.642} C_VEL
LIN {X 0,Y 531.357,Z 135.846,A -85,B 0,C 180,E1 21023.21,E2 21023.21} C_VEL
LIN {X 0,Y 528.72,Z 136.188,A -85,B 0,C 180,E1 21022.095,E2 21022.095} C_VEL
LIN {X 0,Y 528.475,Z 136.22,A -85,B 0,C 180,E1 21021.672,E2 21021.672} C_VEL
LIN {X 0,Y 528.448,Z 136.221,A -85,B 0,C 180,E1 21018.361,E2 21018.361} C_VEL
LIN {X 0,Y 528.49,Z 136.203,A -85,B 0,C 180,E1 21015.036,E2 21015.036} C_VEL
LIN {X 0,Y 528.504,Z 136.517,A -85,B 0,C 180,E1 21013.791,E2 21013.791} C_VEL
LIN {X 0,Y 530.114,Z 140.1,A -85,B 0,C 180,E1 21013.277,E2 21013.277} C_VEL
LIN {X 0,Y 537.891,Z 156.744,A -85,B 0,C 180,E1 21011.149,E2 21011.149} C_VEL
LIN {X 0,Y 541.003,Z 163.784,A -85,B 0,C 180,E1 21010.303,E2 21010.303} C_VEL
LIN {X 0,Y 539.055,Z 208.257,A -85,B 0,C 180,E1 21007.138,E2 21007.138} C_VEL
LIN {X 0,Y 541.66,Z 224.797,A -85,B 0,C 180,E1 21006.626,E2 21006.626} C_VEL
LIN {X 0,Y 539.21,Z 457.017,A -85,B 0,C 180,E1 21003.12,E2 21003.12} C_VEL
LIN {X 0,Y 538.531,Z 516.194,A -85,B 0,C 180,E1 21002.209,E2 21002.209} C_VEL
LIN {X 0,Y 537.868,Z 537.825,A -85,B 0,C 180,E1 21001.679,E2 21001.679} C_VEL
LIN {X 0,Y 537.119,Z 559.413,A -85,B 0,C 180,E1 21000.946,E2 21000.946} C_VEL
LIN {X 0,Y 536.248,Z 579.059,A -85,B 0,C 180,E1 21000.1,E2 21000.1} C_VEL
LIN {X 0,Y 535.262,Z 598.669,A -85,B 0,C 180,E1 20999.048,E2 20999.048} C_VEL
LIN {X 0,Y 534.119,Z 619.235,A -85,B 0,C 180,E1 20997.721,E2 20997.721} C_VEL
LIN {X 0,Y 533.058,Z 638.11,A -85,B 0,C 180,E1 20996.273,E2 20996.273} C_VEL
LIN {X 0,Y 531.999,Z 655.956,A -85,B 0,C 180,E1 20994.659,E2 20994.659} C_VEL
LIN {X 0,Y 531.041,Z 672.293,A -85,B 0,C 180,E1 20992.938,E2 20992.938} C_VEL
LIN {X 0,Y 530.174,Z 688.197,A -85,B 0,C 180,E1 20990.997,E2 20990.997} C_VEL
LIN {X 0,Y 529.516,Z 701.841,A -85,B 0,C 180,E1 20989.066,E2 20989.066} C_VEL
LIN {X 0,Y 528.933,Z 714.71,A -85,B 0,C 180,E1 20986.924,E2 20986.924} C_VEL
LIN {X 0,Y 528.504,Z 726.112,A -85,B 0,C 180,E1 20984.685,E2 20984.685} C_VEL
LIN {X 0,Y 528.229,Z 735.591,A -85,B 0,C 180,E1 20982.461,E2 20982.461} C_VEL
LIN {X 0,Y 528.062,Z 743.239,A -85,B 0,C 180,E1 20980.252,E2 20980.252} C_VEL
LIN {X 0,Y 527.971,Z 749.588,A -85,B 0,C 180,E1 20977.926,E2 20977.926} C_VEL
LIN {X 0,Y 527.928,Z 754.251,A -85,B 0,C 180,E1 20975.652,E2 20975.652} C_VEL
LIN {X 0,Y 527.915,Z 757.239,A -85,B 0,C 180,E1 20973.366,E2 20973.366} C_VEL
LIN {X 0,Y 527.912,Z 758.794,A -85,B 0,C 180,E1 20970.977,E2 20970.977} C_VEL
LIN {X 0,Y 527.911,Z 758.746,A -85,B 0,C 180,E1 20968.698,E2 20968.698} C_VEL
LIN {X 0,Y 527.914,Z 757.108,A -85,B 0,C 180,E1 20966.417,E2 20966.417} C_VEL
LIN {X 0,Y 527.932,Z 754.013,A -85,B 0,C 180,E1 20964.13,E2 20964.13} C_VEL
LIN {X 0,Y 527.974,Z 749.496,A -85,B 0,C 180,E1 20961.944,E2 20961.944} C_VEL
LIN {X 0,Y 528.064,Z 742.821,A -85,B 0,C 180,E1 20959.527,E2 20959.527} C_VEL
LIN {X 0,Y 528.241,Z 735.105,A -85,B 0,C 180,E1 20957.317,E2 20957.317} C_VEL
LIN {X 0,Y 528.521,Z 725.49,A -85,B 0,C 180,E1 20955.091,E2 20955.091} C_VEL
LIN {X 0,Y 528.955,Z 713.945,A -85,B 0,C 180,E1 20952.85,E2 20952.85} C_VEL
LIN {X 0,Y 529.542,Z 701.194,A -85,B 0,C 180,E1 20950.749,E2 20950.749} C_VEL
LIN {X 0,Y 530.239,Z 687.155,A -85,B 0,C 180,E1 20948.774,E2 20948.774} C_VEL
LIN {X 0,Y 531.088,Z 671.51,A -85,B 0,C 180,E1 20946.883,E2 20946.883} C_VEL
LIN {X 0,Y 532.105,Z 653.858,A -85,B 0,C 180,E1 20945.049,E2 20945.049} C_VEL
LIN {X 0,Y 533.197,Z 635.734,A -85,B 0,C 180,E1 20943.442,E2 20943.442} C_VEL
LIN {X 0,Y 534.243,Z 617.306,A -85,B 0,C 180,E1 20942.052,E2 20942.052} C_VEL
LIN {X 0,Y 535.295,Z 598.005,A -85,B 0,C 180,E1 20940.824,E2 20940.824} C_VEL
LIN {X 0,Y 536.289,Z 578.327,A -85,B 0,C 180,E1 20939.777,E2 20939.777} C_VEL
LIN {X 0,Y 537.16,Z 558.429,A -85,B 0,C 180,E1 20938.925,E2 20938.925} C_VEL
LIN {X 0,Y 537.922,Z 536.213,A -85,B 0,C 180,E1 20938.186,E2 20938.186} C_VEL
LIN {X 0,Y 538.555,Z 514.768,A -85,B 0,C 180,E1 20937.675,E2 20937.675} C_VEL
LIN {X 0,Y 540.882,Z 295.278,A -85,B 0,C 180,E1 20934.358,E2 20934.358} C_VEL
LIN {X 0,Y 541.504,Z 222.721,A -85,B 0,C 180,E1 20933.238,E2 20933.238} C_VEL
LIN {X 0,Y 539.054,Z 208.632,A -85,B 0,C 180,E1 20932.796,E2 20932.796} C_VEL
LIN {X 0,Y 541.028,Z 163.794,A -85,B 0,C 180,E1 20929.609,E2 20929.609} C_VEL
LIN {X 0,Y 533.992,Z 148.24,A -85,B 0,C 180,E1 20927.698,E2 20927.698} C_VEL
LIN {X 0,Y 529.913,Z 139.823,A -85,B 0,C 180,E1 20926.588,E2 20926.588} C_VEL
LIN {X 0,Y 528.509,Z 136.52,A -85,B 0,C 180,E1 20926.12,E2 20926.12} C_VEL
LIN {X 0,Y 528.493,Z 136.204,A -85,B 0,C 180,E1 20924.964,E2 20924.964} C_VEL
LIN {X 0,Y 528.446,Z 136.222,A -85,B 0,C 180,E1 20921.639,E2 20921.639} C_VEL
LIN {X 0,Y 528.478,Z 136.221,A -85,B 0,C 180,E1 20918.357,E2 20918.357} C_VEL
LIN {X 0,Y 528.473,Z 136.198,A -85,B 0,C 180,E1 20915.111,E2 20915.111} C_VEL
LIN {X 0,Y 528.45,Z 136.21,A -85,B 0,C 180,E1 20911.842,E2 20911.842} C_VEL
LIN {X 0,Y 528.516,Z 136.216,A -85,B 0,C 180,E1 20908.596,E2 20908.596} C_VEL
LIN {X 0,Y 528.47,Z 136.196,A -85,B 0,C 180,E1 20905.265,E2 20905.265} C_VEL
LIN {X 0,Y 528.461,Z 136.217,A -85,B 0,C 180,E1 20901.884,E2 20901.884} C_VEL
LIN {X 0,Y 528.517,Z 136.193,A -85,B 0,C 180,E1 20898.599,E2 20898.599} C_VEL
LIN {X 0,Y 528.482,Z 136.218,A -85,B 0,C 180,E1 20895.247,E2 20895.247} C_VEL
LIN {X 0,Y 528.472,Z 136.214,A -85,B 0,C 180,E1 20891.901,E2 20891.901} C_VEL
LIN {X 0,Y 528.526,Z 136.21,A -85,B 0,C 180,E1 20888.595,E2 20888.595} C_VEL
LIN {X 0,Y 528.489,Z 136.217,A -85,B 0,C 180,E1 20885.319,E2 20885.319} C_VEL
LIN {X 0,Y 528.479,Z 136.215,A -85,B 0,C 180,E1 20881.843,E2 20881.843} C_VEL
LIN {X 0,Y 528.522,Z 136.212,A -85,B 0,C 180,E1 20878.482,E2 20878.482} C_VEL
LIN {X 0,Y 528.519,Z 136.216,A -85,B 0,C 180,E1 20875.008,E2 20875.008} C_VEL
LIN {X 0,Y 528.487,Z 136.213,A -85,B 0,C 180,E1 20871.624,E2 20871.624} C_VEL
LIN {X 0,Y 528.508,Z 136.21,A -85,B 0,C 180,E1 20868.21,E2 20868.21} C_VEL
LIN {X 0,Y 528.524,Z 136.188,A -85,B 0,C 180,E1 20864.867,E2 20864.867} C_VEL
LIN {X 0,Y 528.504,Z 136.215,A -85,B 0,C 180,E1 20861.405,E2 20861.405} C_VEL
LIN {X 0,Y 528.499,Z 136.192,A -85,B 0,C 180,E1 20857.971,E2 20857.971} C_VEL
LIN {X 0,Y 528.524,Z 136.206,A -85,B 0,C 180,E1 20854.568,E2 20854.568} C_VEL
LIN {X 0,Y 528.524,Z 136.208,A -85,B 0,C 180,E1 20851.034,E2 20851.034} C_VEL
LIN {X 0,Y 528.503,Z 136.195,A -85,B 0,C 180,E1 20847.629,E2 20847.629} C_VEL
LIN {X 0,Y 528.522,Z 136.205,A -85,B 0,C 180,E1 20844.228,E2 20844.228} C_VEL
LIN {X 0,Y 528.515,Z 136.212,A -85,B 0,C 180,E1 20840.812,E2 20840.812} C_VEL
LIN {X 0,Y 528.518,Z 136.216,A -85,B 0,C 180,E1 20837.37,E2 20837.37} C_VEL
LIN {X 0,Y 528.545,Z 136.37,A -85,B 0,C 180,E1 20836.182,E2 20836.182} C_VEL
LIN {X 0,Y 529.11,Z 138.382,A -85,B 0,C 180,E1 20835.895,E2 20835.895} C_VEL
LIN {X 0,Y 530.913,Z 141.676,A -85,B 0,C 180,E1 20835.451,E2 20835.451} C_VEL
LIN {X 0,Y 541.092,Z 162.063,A -85,B 0,C 180,E1 20832.967,E2 20832.967} C_VEL
LIN {X 0,Y 543.919,Z 166.705,A -85,B 0,C 180,E1 20832.629,E2 20832.629} C_VEL
LIN {X 0,Y 546.007,Z 179.423,A -85,B 0,C 180,E1 20832.206,E2 20832.206} C_VEL
LIN {X 0,Y 543.376,Z 385.998,A -85,B 0,C 180,E1 20828.93,E2 20828.93} C_VEL
LIN {X 0,Y 541.802,Z 511.393,A -85,B 0,C 180,E1 20826.961,E2 20826.961} C_VEL
LIN {X 0,Y 541.067,Z 534.527,A -85,B 0,C 180,E1 20826.411,E2 20826.411} C_VEL
LIN {X 0,Y 540.184,Z 556.135,A -85,B 0,C 180,E1 20825.717,E2 20825.717} C_VEL
LIN {X 0,Y 539.159,Z 577.415,A -85,B 0,C 180,E1 20824.831,E2 20824.831} C_VEL
LIN {X 0,Y 538.073,Z 597.209,A -85,B 0,C 180,E1 20823.837,E2 20823.837} C_VEL
LIN {X 0,Y 536.754,Z 618.259,A -85,B 0,C 180,E1 20822.57,E2 20822.57} C_VEL
LIN {X 0,Y 535.49,Z 638.422,A -85,B 0,C 180,E1 20821.144,E2 20821.144} C_VEL
LIN {X 0,Y 534.111,Z 658.284,A -85,B 0,C 180,E1 20819.493,E2 20819.493} C_VEL
LIN {X 0,Y 532.814,Z 677.798,A -85,B 0,C 180,E1 20817.613,E2 20817.613} C_VEL
LIN {X 0,Y 531.722,Z 694.667,A -85,B 0,C 180,E1 20815.745,E2 20815.745} C_VEL
LIN {X 0,Y 530.696,Z 710.999,A -85,B 0,C 180,E1 20813.659,E2 20813.659} C_VEL
LIN {X 0,Y 529.869,Z 725.93,A -85,B 0,C 180,E1 20811.473,E2 20811.473} C_VEL
LIN {X 0,Y 529.229,Z 738.732,A -85,B 0,C 180,E1 20809.306,E2 20809.306} C_VEL
LIN {X 0,Y 528.699,Z 751.054,A -85,B 0,C 180,E1 20806.878,E2 20806.878} C_VEL
LIN {X 0,Y 528.365,Z 760.992,A -85,B 0,C 180,E1 20804.577,E2 20804.577} C_VEL
LIN {X 0,Y 528.131,Z 769.701,A -85,B 0,C 180,E1 20802.131,E2 20802.131} C_VEL
LIN {X 0,Y 527.996,Z 776.474,A -85,B 0,C 180,E1 20799.813,E2 20799.813} C_VEL
LIN {X 0,Y 527.941,Z 781.841,A -85,B 0,C 180,E1 20797.399,E2 20797.399} C_VEL
LIN {X 0,Y 527.919,Z 785.596,A -85,B 0,C 180,E1 20795.107,E2 20795.107} C_VEL
LIN {X 0,Y 527.913,Z 788.056,A -85,B 0,C 180,E1 20792.605,E2 20792.605} C_VEL
LIN {X 0,Y 527.9,Z 788.939,A -85,B 0,C 180,E1 20790.326,E2 20790.326} C_VEL
LIN {X 0,Y 527.907,Z 788.324,A -85,B 0,C 180,E1 20787.829,E2 20787.829} C_VEL
LIN {X 0,Y 527.902,Z 786.503,A -85,B 0,C 180,E1 20785.655,E2 20785.655} C_VEL
LIN {X 0,Y 527.939,Z 782.668,A -85,B 0,C 180,E1 20783.038,E2 20783.038} C_VEL
LIN {X 0,Y 527.987,Z 778.063,A -85,B 0,C 180,E1 20780.847,E2 20780.847} C_VEL
LIN {X 0,Y 528.106,Z 771.118,A -85,B 0,C 180,E1 20778.312,E2 20778.312} C_VEL
LIN {X 0,Y 528.281,Z 763.524,A -85,B 0,C 180,E1 20776.092,E2 20776.092} C_VEL
LIN {X 0,Y 528.611,Z 753.399,A -85,B 0,C 180,E1 20773.631,E2 20773.631} C_VEL
LIN {X 0,Y 529.052,Z 742.41,A -85,B 0,C 180,E1 20771.374,E2 20771.374} C_VEL
LIN {X 0,Y 529.668,Z 729.465,A -85,B 0,C 180,E1 20769.098,E2 20769.098} C_VEL
LIN {X 0,Y 530.477,Z 715.058,A -85,B 0,C 180,E1 20766.896,E2 20766.896} C_VEL
LIN {X 0,Y 531.405,Z 699.335,A -85,B 0,C 180,E1 20764.825,E2 20764.825} C_VEL
LIN {X 0,Y 532.58,Z 681.126,A -85,B 0,C 180,E1 20762.737,E2 20762.737} C_VEL
LIN {X 0,Y 533.838,Z 662.911,A -85,B 0,C 180,E1 20760.921,E2 20760.921} C_VEL
LIN {X 0,Y 535.096,Z 643.572,A -85,B 0,C 180,E1 20759.264,E2 20759.264} C_VEL
LIN {X 0,Y 536.496,Z 622.743,A -85,B 0,C 180,E1 20757.729,E2 20757.729} C_VEL
LIN {X 0,Y 537.71,Z 602.832,A -85,B 0,C 180,E1 20756.479,E2 20756.479} C_VEL
LIN {X 0,Y 538.959,Z 581.269,A -85,B 0,C 180,E1 20755.348,E2 20755.348} C_VEL
LIN {X 0,Y 539.933,Z 562.005,A -85,B 0,C 180,E1 20754.512,E2 20754.512} C_VEL
LIN {X 0,Y 540.905,Z 538.392,A -85,B 0,C 180,E1 20753.698,E2 20753.698} C_VEL
LIN {X 0,Y 541.646,Z 516.969,A -85,B 0,C 180,E1 20753.152,E2 20753.152} C_VEL
LIN {X 0,Y 542.204,Z 484.974,A -85,B 0,C 180,E1 20752.604,E2 20752.604} C_VEL
LIN {X 0,Y 544.749,Z 275.38,A -85,B 0,C 180,E1 20749.329,E2 20749.329} C_VEL
LIN {X 0,Y 545.873,Z 177.518,A -85,B 0,C 180,E1 20747.748,E2 20747.748} C_VEL
LIN {X 0,Y 543.537,Z 165.744,A -85,B 0,C 180,E1 20747.318,E2 20747.318} C_VEL
LIN {X 0,Y 540.569,Z 161.002,A -85,B 0,C 180,E1 20746.937,E2 20746.937} C_VEL
LIN {X 0,Y 530.321,Z 140.348,A -85,B 0,C 180,E1 20744.385,E2 20744.385} C_VEL
LIN {X 0,Y 528.622,Z 136.825,A -85,B 0,C 180,E1 20743.919,E2 20743.919} C_VEL
LIN {X 0,Y 528.521,Z 136.201,A -85,B 0,C 180,E1 20743.67,E2 20743.67} C_VEL
LIN {X 0,Y 528.508,Z 136.197,A -85,B 0,C 180,E1 20740.317,E2 20740.317} C_VEL
LIN {X 0,Y 528.518,Z 136.194,A -85,B 0,C 180,E1 20736.984,E2 20736.984} C_VEL
LIN {X 0,Y 528.52,Z 136.204,A -85,B 0,C 180,E1 20733.461,E2 20733.461} C_VEL
LIN {X 0,Y 528.506,Z 136.213,A -85,B 0,C 180,E1 20730.089,E2 20730.089} C_VEL
LIN {X 0,Y 528.51,Z 136.197,A -85,B 0,C 180,E1 20726.639,E2 20726.639} C_VEL
LIN {X 0,Y 528.523,Z 136.205,A -85,B 0,C 180,E1 20723.172,E2 20723.172} C_VEL
LIN {X 0,Y 528.519,Z 136.205,A -85,B 0,C 180,E1 20719.678,E2 20719.678} C_VEL
LIN {X 0,Y 528.493,Z 136.196,A -85,B 0,C 180,E1 20716.26,E2 20716.26} C_VEL
LIN {X 0,Y 528.52,Z 136.21,A -85,B 0,C 180,E1 20712.899,E2 20712.899} C_VEL
LIN {X 0,Y 528.524,Z 136.206,A -85,B 0,C 180,E1 20709.473,E2 20709.473} C_VEL
LIN {X 0,Y 528.487,Z 136.212,A -85,B 0,C 180,E1 20706.191,E2 20706.191} C_VEL
LIN {X 0,Y 528.509,Z 136.213,A -85,B 0,C 180,E1 20702.819,E2 20702.819} C_VEL
LIN {X 0,Y 528.529,Z 136.205,A -85,B 0,C 180,E1 20699.458,E2 20699.458} C_VEL
LIN {X 0,Y 528.481,Z 136.208,A -85,B 0,C 180,E1 20696.094,E2 20696.094} C_VEL
LIN {X 0,Y 528.487,Z 136.212,A -85,B 0,C 180,E1 20692.608,E2 20692.608} C_VEL
LIN {X 0,Y 528.525,Z 136.21,A -85,B 0,C 180,E1 20689.316,E2 20689.316} C_VEL
LIN {X 0,Y 528.477,Z 136.211,A -85,B 0,C 180,E1 20685.985,E2 20685.985} C_VEL
LIN {X 0,Y 528.471,Z 136.208,A -85,B 0,C 180,E1 20682.465,E2 20682.465} C_VEL
LIN {X 0,Y 528.526,Z 136.201,A -85,B 0,C 180,E1 20679.15,E2 20679.15} C_VEL
LIN {X 0,Y 528.475,Z 136.21,A -85,B 0,C 180,E1 20675.879,E2 20675.879} C_VEL
LIN {X 0,Y 528.465,Z 136.218,A -85,B 0,C 180,E1 20672.506,E2 20672.506} C_VEL
LIN {X 0,Y 528.521,Z 136.193,A -85,B 0,C 180,E1 20669.188,E2 20669.188} C_VEL
LIN {X 0,Y 528.462,Z 136.218,A -85,B 0,C 180,E1 20665.941,E2 20665.941} C_VEL
LIN {X 0,Y 528.452,Z 136.221,A -85,B 0,C 180,E1 20662.443,E2 20662.443} C_VEL
LIN {X 0,Y 528.475,Z 136.22,A -85,B 0,C 180,E1 20661.672,E2 20661.672} C_VEL
LIN {X 0,Y 527.525,Z 136.343,A -85,B 0,C 180,E1 20660.836,E2 20660.836} C_VEL
LIN {X 0,Y 521.032,Z 137.145,A -85,B 0,C 180,E1 20658.489,E2 20658.489} C_VEL
LIN {X 0,Y 520.519,Z 137.211,A -85,B 0,C 180,E1 20657.877,E2 20657.877} C_VEL
LIN {X 0,Y 520.536,Z 137.355,A -85,B 0,C 180,E1 20654.637,E2 20654.637} C_VEL
LIN {X 0,Y 520.963,Z 139.056,A -85,B 0,C 180,E1 20654.363,E2 20654.363} C_VEL
LIN {X 0,Y 523.185,Z 143.411,A -85,B 0,C 180,E1 20653.747,E2 20653.747} C_VEL
LIN {X 0,Y 530.132,Z 157.69,A -85,B 0,C 180,E1 20651.841,E2 20651.841} C_VEL
LIN {X 0,Y 534.463,Z 167.715,A -85,B 0,C 180,E1 20650.618,E2 20650.618} C_VEL
LIN {X 0,Y 532.436,Z 208.525,A -85,B 0,C 180,E1 20647.68,E2 20647.68} C_VEL
LIN {X 0,Y 535.226,Z 226.34,A -85,B 0,C 180,E1 20647.115,E2 20647.115} C_VEL
LIN {X 0,Y 532.498,Z 458.607,A -85,B 0,C 180,E1 20643.568,E2 20643.568} C_VEL
LIN {X 0,Y 531.756,Z 516.402,A -85,B 0,C 180,E1 20642.666,E2 20642.666} C_VEL
LIN {X 0,Y 531.033,Z 538.058,A -85,B 0,C 180,E1 20642.129,E2 20642.129} C_VEL
LIN {X 0,Y 530.204,Z 559.429,A -85,B 0,C 180,E1 20641.395,E2 20641.395} C_VEL
LIN {X 0,Y 529.219,Z 579.679,A -85,B 0,C 180,E1 20640.511,E2 20640.511} C_VEL
LIN {X 0,Y 528.112,Z 599.378,A -85,B 0,C 180,E1 20639.436,E2 20639.436} C_VEL
LIN {X 0,Y 526.878,Z 619.416,A -85,B 0,C 180,E1 20638.123,E2 20638.123} C_VEL
LIN {X 0,Y 525.702,Z 638.115,A -85,B 0,C 180,E1 20636.67,E2 20636.67} C_VEL
LIN {X 0,Y 524.516,Z 655.965,A -85,B 0,C 180,E1 20635.035,E2 20635.035} C_VEL
LIN {X 0,Y 523.432,Z 672.665,A -85,B 0,C 180,E1 20633.248,E2 20633.248} C_VEL
LIN {X 0,Y 522.448,Z 688.738,A -85,B 0,C 180,E1 20631.248,E2 20631.248} C_VEL
LIN {X 0,Y 521.692,Z 702.57,A -85,B 0,C 180,E1 20629.247,E2 20629.247} C_VEL
LIN {X 0,Y 521.059,Z 715.004,A -85,B 0,C 180,E1 20627.135,E2 20627.135} C_VEL
LIN {X 0,Y 520.583,Z 726.116,A -85,B 0,C 180,E1 20624.913,E2 20624.913} C_VEL
LIN {X 0,Y 520.271,Z 735.595,A -85,B 0,C 180,E1 20622.655,E2 20622.655} C_VEL
LIN {X 0,Y 520.08,Z 743.241,A -85,B 0,C 180,E1 20620.411,E2 20620.411} C_VEL
LIN {X 0,Y 519.979,Z 749.719,A -85,B 0,C 180,E1 20617.992,E2 20617.992} C_VEL
LIN {X 0,Y 519.928,Z 754.418,A -85,B 0,C 180,E1 20615.628,E2 20615.628} C_VEL
LIN {X 0,Y 519.915,Z 757.353,A -85,B 0,C 180,E1 20613.307,E2 20613.307} C_VEL
LIN {X 0,Y 519.908,Z 758.817,A -85,B 0,C 180,E1 20610.882,E2 20610.882} C_VEL
LIN {X 0,Y 519.906,Z 758.723,A -85,B 0,C 180,E1 20608.567,E2 20608.567} C_VEL
LIN {X 0,Y 519.914,Z 756.995,A -85,B 0,C 180,E1 20606.251,E2 20606.251} C_VEL
LIN {X 0,Y 519.933,Z 753.601,A -85,B 0,C 180,E1 20603.818,E2 20603.818} C_VEL
LIN {X 0,Y 519.978,Z 748.986,A -85,B 0,C 180,E1 20601.597,E2 20601.597} C_VEL
LIN {X 0,Y 520.089,Z 742.395,A -85,B 0,C 180,E1 20599.231,E2 20599.231} C_VEL
LIN {X 0,Y 520.302,Z 734.559,A -85,B 0,C 180,E1 20596.982,E2 20596.982} C_VEL
LIN {X 0,Y 520.626,Z 724.968,A -85,B 0,C 180,E1 20594.746,E2 20594.746} C_VEL
LIN {X 0,Y 521.126,Z 713.304,A -85,B 0,C 180,E1 20592.469,E2 20592.469} C_VEL
LIN {X 0,Y 521.773,Z 700.901,A -85,B 0,C 180,E1 20590.407,E2 20590.407} C_VEL
LIN {X 0,Y 522.569,Z 686.937,A -85,B 0,C 180,E1 20588.418,E2 20588.418} C_VEL
LIN {X 0,Y 523.508,Z 671.547,A -85,B 0,C 180,E1 20586.534,E2 20586.534} C_VEL
LIN {X 0,Y 524.644,Z 653.848,A -85,B 0,C 180,E1 20584.67,E2 20584.67} C_VEL
LIN {X 0,Y 525.82,Z 636.365,A -85,B 0,C 180,E1 20583.093,E2 20583.093} C_VEL
LIN {X 0,Y 526.979,Z 617.99,A -85,B 0,C 180,E1 20581.685,E2 20581.685} C_VEL
LIN {X 0,Y 528.184,Z 597.988,A -85,B 0,C 180,E1 20580.392,E2 20580.392} C_VEL
LIN {X 0,Y 529.298,Z 578.315,A -85,B 0,C 180,E1 20579.335,E2 20579.335} C_VEL
LIN {X 0,Y 530.265,Z 558.075,A -85,B 0,C 180,E1 20578.461,E2 20578.461} C_VEL
LIN {X 0,Y 531.106,Z 536.145,A -85,B 0,C 180,E1 20577.727,E2 20577.727} C_VEL
LIN {X 0,Y 531.789,Z 514.69,A -85,B 0,C 180,E1 20577.212,E2 20577.212} C_VEL
LIN {X 0,Y 534.364,Z 296.627,A -85,B 0,C 180,E1 20573.878,E2 20573.878} C_VEL
LIN {X 0,Y 535.071,Z 224.201,A -85,B 0,C 180,E1 20572.747,E2 20572.747} C_VEL
LIN {X 0,Y 532.429,Z 208.311,A -85,B 0,C 180,E1 20572.218,E2 20572.218} C_VEL
LIN {X 0,Y 534.434,Z 167.386,A -85,B 0,C 180,E1 20569.262,E2 20569.262} C_VEL
LIN {X 0,Y 527.464,Z 152.194,A -85,B 0,C 180,E1 20567.349,E2 20567.349} C_VEL
LIN {X 0,Y 522.27,Z 141.295,A -85,B 0,C 180,E1 20565.883,E2 20565.883} C_VEL
LIN {X 0,Y 520.592,Z 137.655,A -85,B 0,C 180,E1 20565.357,E2 20565.357} C_VEL
LIN {X 0,Y 520.552,Z 137.192,A -85,B 0,C 180,E1 20564.979,E2 20564.979} C_VEL
LIN {X 0,Y 520.508,Z 137.211,A -85,B 0,C 180,E1 20561.65,E2 20561.65} C_VEL
LIN {X 0,Y 520.537,Z 137.209,A -85,B 0,C 180,E1 20558.347,E2 20558.347} C_VEL
LIN {X 0,Y 520.54,Z 137.185,A -85,B 0,C 180,E1 20555.052,E2 20555.052} C_VEL
LIN {X 0,Y 520.509,Z 137.196,A -85,B 0,C 180,E1 20551.758,E2 20551.758} C_VEL
LIN {X 0,Y 520.558,Z 137.207,A -85,B 0,C 180,E1 20548.447,E2 20548.447} C_VEL
LIN {X 0,Y 520.543,Z 137.181,A -85,B 0,C 180,E1 20545.119,E2 20545.119} C_VEL
LIN {X 0,Y 520.521,Z 137.206,A -85,B 0,C 180,E1 20541.761,E2 20541.761} C_VEL
LIN {X 0,Y 520.561,Z 137.184,A -85,B 0,C 180,E1 20538.411,E2 20538.411} C_VEL
LIN {X 0,Y 520.564,Z 137.204,A -85,B 0,C 180,E1 20535.029,E2 20535.029} C_VEL
LIN {X 0,Y 520.532,Z 137.204,A -85,B 0,C 180,E1 20531.636,E2 20531.636} C_VEL
LIN {X 0,Y 520.549,Z 137.2,A -85,B 0,C 180,E1 20528.172,E2 20528.172} C_VEL
LIN {X 0,Y 520.585,Z 137.2,A -85,B 0,C 180,E1 20524.848,E2 20524.848} C_VEL
LIN {X 0,Y 520.547,Z 137.205,A -85,B 0,C 180,E1 20521.431,E2 20521.431} C_VEL
LIN {X 0,Y 520.546,Z 137.203,A -85,B 0,C 180,E1 20517.909,E2 20517.909} C_VEL
LIN {X 0,Y 520.583,Z 137.199,A -85,B 0,C 180,E1 20514.489,E2 20514.489} C_VEL
LIN {X 0,Y 520.582,Z 137.203,A -85,B 0,C 180,E1 20511.05,E2 20511.05} C_VEL
LIN {X 0,Y 520.554,Z 137.203,A -85,B 0,C 180,E1 20507.577,E2 20507.577} C_VEL
LIN {X 0,Y 520.56,Z 137.18,A -85,B 0,C 180,E1 20504.058,E2 20504.058} C_VEL
LIN {X 0,Y 520.585,Z 137.197,A -85,B 0,C 180,E1 20500.71,E2 20500.71} C_VEL
LIN {X 0,Y 520.58,Z 137.185,A -85,B 0,C 180,E1 20497.172,E2 20497.172} C_VEL
LIN {X 0,Y 520.56,Z 137.192,A -85,B 0,C 180,E1 20493.761,E2 20493.761} C_VEL
LIN {X 0,Y 520.588,Z 137.2,A -85,B 0,C 180,E1 20490.296,E2 20490.296} C_VEL
LIN {X 0,Y 520.579,Z 137.186,A -85,B 0,C 180,E1 20486.812,E2 20486.812} C_VEL
LIN {X 0,Y 520.577,Z 137.181,A -85,B 0,C 180,E1 20483.321,E2 20483.321} C_VEL
LIN {X 0,Y 520.572,Z 137.185,A -85,B 0,C 180,E1 20479.855,E2 20479.855} C_VEL
LIN {X 0,Y 520.592,Z 137.295,A -85,B 0,C 180,E1 20477.014,E2 20477.014} C_VEL
LIN {X 0,Y 520.962,Z 138.846,A -85,B 0,C 180,E1 20476.751,E2 20476.751} C_VEL
LIN {X 0,Y 523.039,Z 142.774,A -85,B 0,C 180,E1 20476.211,E2 20476.211} C_VEL
LIN {X 0,Y 533.149,Z 162.822,A -85,B 0,C 180,E1 20473.681,E2 20473.681} C_VEL
LIN {X 0,Y 538.267,Z 170.992,A -85,B 0,C 180,E1 20473.064,E2 20473.064} C_VEL
LIN {X 0,Y 539.96,Z 181.054,A -85,B 0,C 180,E1 20472.74,E2 20472.74} C_VEL
LIN {X 0,Y 537.188,Z 383.58,A -85,B 0,C 180,E1 20469.506,E2 20469.506} C_VEL
LIN {X 0,Y 535.404,Z 511.378,A -85,B 0,C 180,E1 20467.478,E2 20467.478} C_VEL
LIN {X 0,Y 534.611,Z 534.394,A -85,B 0,C 180,E1 20466.927,E2 20466.927} C_VEL
LIN {X 0,Y 533.661,Z 555.492,A -85,B 0,C 180,E1 20466.248,E2 20466.248} C_VEL
LIN {X 0,Y 532.489,Z 577.412,A -85,B 0,C 180,E1 20465.332,E2 20465.332} C_VEL
LIN {X 0,Y 531.275,Z 597.594,A -85,B 0,C 180,E1 20464.308,E2 20464.308} C_VEL
LIN {X 0,Y 529.772,Z 619.155,A -85,B 0,C 180,E1 20462.989,E2 20462.989} C_VEL
LIN {X 0,Y 528.372,Z 639.198,A -85,B 0,C 180,E1 20461.548,E2 20461.548} C_VEL
LIN {X 0,Y 526.898,Z 658.281,A -85,B 0,C 180,E1 20459.938,E2 20459.938} C_VEL
LIN {X 0,Y 525.422,Z 678.141,A -85,B 0,C 180,E1 20457.997,E2 20457.997} C_VEL
LIN {X 0,Y 524.218,Z 694.667,A -85,B 0,C 180,E1 20456.141,E2 20456.141} C_VEL
LIN {X 0,Y 523.068,Z 710.997,A -85,B 0,C 180,E1 20454.026,E2 20454.026} C_VEL
LIN {X 0,Y 522.12,Z 726.244,A -85,B 0,C 180,E1 20451.756,E2 20451.756} C_VEL
LIN {X 0,Y 521.407,Z 738.73,A -85,B 0,C 180,E1 20449.607,E2 20449.607} C_VEL
LIN {X 0,Y 520.818,Z 750.807,A -85,B 0,C 180,E1 20447.196,E2 20447.196} C_VEL
LIN {X 0,Y 520.436,Z 760.587,A -85,B 0,C 180,E1 20444.904,E2 20444.904} C_VEL
LIN {X 0,Y 520.173,Z 769.346,A -85,B 0,C 180,E1 20442.432,E2 20442.432} C_VEL
LIN {X 0,Y 520.029,Z 776.031,A -85,B 0,C 180,E1 20440.128,E2 20440.128} C_VEL
LIN {X 0,Y 519.952,Z 781.635,A -85,B 0,C 180,E1 20437.625,E2 20437.625} C_VEL
LIN {X 0,Y 519.911,Z 785.277,A -85,B 0,C 180,E1 20435.407,E2 20435.407} C_VEL
LIN {X 0,Y 519.916,Z 787.987,A -85,B 0,C 180,E1 20432.756,E2 20432.756} C_VEL
LIN {X 0,Y 519.898,Z 788.917,A -85,B 0,C 180,E1 20430.441,E2 20430.441} C_VEL
LIN {X 0,Y 519.908,Z 788.392,A -85,B 0,C 180,E1 20427.906,E2 20427.906} C_VEL
LIN {X 0,Y 519.904,Z 786.616,A -85,B 0,C 180,E1 20425.699,E2 20425.699} C_VEL
LIN {X 0,Y 519.939,Z 783.081,A -85,B 0,C 180,E1 20423.153,E2 20423.153} C_VEL
LIN {X 0,Y 519.988,Z 778.573,A -85,B 0,C 180,E1 20420.928,E2 20420.928} C_VEL
LIN {X 0,Y 520.114,Z 772.177,A -85,B 0,C 180,E1 20418.468,E2 20418.468} C_VEL
LIN {X 0,Y 520.318,Z 764.081,A -85,B 0,C 180,E1 20416.029,E2 20416.029} C_VEL
LIN {X 0,Y 520.694,Z 753.912,A -85,B 0,C 180,E1 20413.49,E2 20413.49} C_VEL
LIN {X 0,Y 521.186,Z 742.992,A -85,B 0,C 180,E1 20411.199,E2 20411.199} C_VEL
LIN {X 0,Y 521.911,Z 729.463,A -85,B 0,C 180,E1 20408.773,E2 20408.773} C_VEL
LIN {X 0,Y 522.814,Z 715.221,A -85,B 0,C 180,E1 20406.561,E2 20406.561} C_VEL
LIN {X 0,Y 523.869,Z 699.416,A -85,B 0,C 180,E1 20404.448,E2 20404.448} C_VEL
LIN {X 0,Y 525.19,Z 681.127,A -85,B 0,C 180,E1 20402.321,E2 20402.321} C_VEL
LIN {X 0,Y 526.587,Z 662.912,A -85,B 0,C 180,E1 20400.481,E2 20400.481} C_VEL
LIN {X 0,Y 527.977,Z 643.9,A -85,B 0,C 180,E1 20398.832,E2 20398.832} C_VEL
LIN {X 0,Y 529.542,Z 622.746,A -85,B 0,C 180,E1 20397.252,E2 20397.252} C_VEL
LIN {X 0,Y 530.899,Z 602.828,A -85,B 0,C 180,E1 20395.99,E2 20395.99} C_VEL
LIN {X 0,Y 532.278,Z 581.266,A -85,B 0,C 180,E1 20394.849,E2 20394.849} C_VEL
LIN {X 0,Y 533.382,Z 561.263,A -85,B 0,C 180,E1 20393.976,E2 20393.976} C_VEL
LIN {X 0,Y 534.458,Z 537.734,A -85,B 0,C 180,E1 20393.168,E2 20393.168} C_VEL
LIN {X 0,Y 535.266,Z 516.319,A -85,B 0,C 180,E1 20392.622,E2 20392.622} C_VEL
LIN {X 0,Y 535.878,Z 482.823,A -85,B 0,C 180,E1 20392.05,E2 20392.05} C_VEL
LIN {X 0,Y 538.707,Z 273.664,A -85,B 0,C 180,E1 20388.744,E2 20388.744} C_VEL
LIN {X 0,Y 539.825,Z 179.241,A -85,B 0,C 180,E1 20387.217,E2 20387.217} C_VEL
LIN {X 0,Y 537.914,Z 170.106,A -85,B 0,C 180,E1 20386.889,E2 20386.889} C_VEL
LIN {X 0,Y 532.765,Z 162.168,A -85,B 0,C 180,E1 20386.265,E2 20386.265} C_VEL
LIN {X 0,Y 524.271,Z 145.236,A -85,B 0,C 180,E1 20384.115,E2 20384.115} C_VEL
LIN {X 0,Y 522.228,Z 141.137,A -85,B 0,C 180,E1 20383.571,E2 20383.571} C_VEL
LIN {X 0,Y 520.623,Z 137.515,A -85,B 0,C 180,E1 20383.058,E2 20383.058} C_VEL
LIN {X 0,Y 520.574,Z 137.196,A -85,B 0,C 180,E1 20382.091,E2 20382.091} C_VEL
LIN {X 0,Y 520.578,Z 137.202,A -85,B 0,C 180,E1 20378.584,E2 20378.584} C_VEL
LIN {X 0,Y 520.581,Z 137.199,A -85,B 0,C 180,E1 20375.097,E2 20375.097} C_VEL
LIN {X 0,Y 520.585,Z 137.184,A -85,B 0,C 180,E1 20371.623,E2 20371.623} C_VEL
LIN {X 0,Y 520.564,Z 137.187,A -85,B 0,C 180,E1 20368.166,E2 20368.166} C_VEL
LIN {X 0,Y 520.572,Z 137.205,A -85,B 0,C 180,E1 20364.632,E2 20364.632} C_VEL
LIN {X 0,Y 520.581,Z 137.176,A -85,B 0,C 180,E1 20361.167,E2 20361.167} C_VEL
LIN {X 0,Y 520.58,Z 137.198,A -85,B 0,C 180,E1 20357.666,E2 20357.666} C_VEL
LIN {X 0,Y 520.553,Z 137.189,A -85,B 0,C 180,E1 20354.232,E2 20354.232} C_VEL
LIN {X 0,Y 520.575,Z 137.198,A -85,B 0,C 180,E1 20350.849,E2 20350.849} C_VEL
LIN {X 0,Y 520.591,Z 137.199,A -85,B 0,C 180,E1 20347.393,E2 20347.393} C_VEL
LIN {X 0,Y 520.554,Z 137.199,A -85,B 0,C 180,E1 20343.965,E2 20343.965} C_VEL
LIN {X 0,Y 520.546,Z 137.199,A -85,B 0,C 180,E1 20340.44,E2 20340.44} C_VEL
LIN {X 0,Y 520.581,Z 137.2,A -85,B 0,C 180,E1 20337.027,E2 20337.027} C_VEL
LIN {X 0,Y 520.572,Z 137.201,A -85,B 0,C 180,E1 20333.604,E2 20333.604} C_VEL
LIN {X 0,Y 520.538,Z 137.203,A -85,B 0,C 180,E1 20330.181,E2 20330.181} C_VEL
LIN {X 0,Y 520.555,Z 137.202,A -85,B 0,C 180,E1 20326.787,E2 20326.787} C_VEL
LIN {X 0,Y 520.582,Z 137.203,A -85,B 0,C 180,E1 20323.411,E2 20323.411} C_VEL
LIN {X 0,Y 520.527,Z 137.186,A -85,B 0,C 180,E1 20320.123,E2 20320.123} C_VEL
LIN {X 0,Y 520.539,Z 137.201,A -85,B 0,C 180,E1 20316.691,E2 20316.691} C_VEL
LIN {X 0,Y 520.58,Z 137.187,A -85,B 0,C 180,E1 20313.292,E2 20313.292} C_VEL
LIN {X 0,Y 520.523,Z 137.196,A -85,B 0,C 180,E1 20310.03,E2 20310.03} C_VEL
LIN {X 0,Y 520.52,Z 137.208,A -85,B 0,C 180,E1 20306.475,E2 20306.475} C_VEL
LIN {X 0,Y 520.572,Z 137.186,A -85,B 0,C 180,E1 20303.183,E2 20303.183} C_VEL
LIN {X 0,Y 520.515,Z 137.188,A -85,B 0,C 180,E1 20299.946,E2 20299.946} C_VEL
LIN {X 0,Y 520.519,Z 137.211,A -85,B 0,C 180,E1 20297.877,E2 20297.877} C_VEL
LIN {X 0,Y 519.714,Z 137.407,A -85,B 0,C 180,E1 20297.372,E2 20297.372} C_VEL
LIN {X 0,Y 513.2,Z 138.096,A -85,B 0,C 180,E1 20295.819,E2 20295.819} C_VEL
LIN {X 0,Y 512.677,Z 138.541,A -85,B 0,C 180,E1 20295.399,E2 20295.399} C_VEL
LIN {X 0,Y 512.706,Z 138.697,A -85,B 0,C 180,E1 20295.366,E2 20295.366} C_VEL
LIN {X 0,Y 514.45,Z 142.404,A -85,B 0,C 180,E1 20294.814,E2 20294.814} C_VEL
LIN {X 0,Y 523.844,Z 161.934,A -85,B 0,C 180,E1 20292.138,E2 20292.138} C_VEL
LIN {X 0,Y 527.914,Z 171.65,A -85,B 0,C 180,E1 20290.942,E2 20290.942} C_VEL
LIN {X 0,Y 525.979,Z 208.555,A -85,B 0,C 180,E1 20288.271,E2 20288.271} C_VEL
LIN {X 0,Y 529.057,Z 227.777,A -85,B 0,C 180,E1 20287.648,E2 20287.648} C_VEL
LIN {X 0,Y 526.283,Z 423.163,A -85,B 0,C 180,E1 20284.593,E2 20284.593} C_VEL
LIN {X 0,Y 525.042,Z 515.701,A -85,B 0,C 180,E1 20283.154,E2 20283.154} C_VEL
LIN {X 0,Y 524.277,Z 537.169,A -85,B 0,C 180,E1 20282.623,E2 20282.623} C_VEL
LIN {X 0,Y 523.324,Z 559.446,A -85,B 0,C 180,E1 20281.856,E2 20281.856} C_VEL
LIN {X 0,Y 522.291,Z 579.045,A -85,B 0,C 180,E1 20280.994,E2 20280.994} C_VEL
LIN {X 0,Y 521.029,Z 599.351,A -85,B 0,C 180,E1 20279.879,E2 20279.879} C_VEL
LIN {X 0,Y 519.694,Z 619.249,A -85,B 0,C 180,E1 20278.56,E2 20278.56} C_VEL
LIN {X 0,Y 518.426,Z 637.452,A -85,B 0,C 180,E1 20277.136,E2 20277.136} C_VEL
LIN {X 0,Y 517.145,Z 654.767,A -85,B 0,C 180,E1 20275.54,E2 20275.54} C_VEL
LIN {X 0,Y 515.911,Z 672.016,A -85,B 0,C 180,E1 20273.686,E2 20273.686} C_VEL
LIN {X 0,Y 514.869,Z 687.36,A -85,B 0,C 180,E1 20271.771,E2 20271.771} C_VEL
LIN {X 0,Y 513.959,Z 701.849,A -85,B 0,C 180,E1 20269.667,E2 20269.667} C_VEL
LIN {X 0,Y 513.248,Z 714.08,A -85,B 0,C 180,E1 20267.575,E2 20267.575} C_VEL
LIN {X 0,Y 512.692,Z 725.601,A -85,B 0,C 180,E1 20265.264,E2 20265.264} C_VEL
LIN {X 0,Y 512.332,Z 735.19,A -85,B 0,C 180,E1 20262.969,E2 20262.969} C_VEL
LIN {X 0,Y 512.104,Z 742.89,A -85,B 0,C 180,E1 20260.689,E2 20260.689} C_VEL
LIN {X 0,Y 511.987,Z 749.545,A -85,B 0,C 180,E1 20258.196,E2 20258.196} C_VEL
LIN {X 0,Y 511.934,Z 754.253,A -85,B 0,C 180,E1 20255.829,E2 20255.829} C_VEL
LIN {X 0,Y 511.913,Z 757.242,A -85,B 0,C 180,E1 20253.471,E2 20253.471} C_VEL
LIN {X 0,Y 511.912,Z 758.794,A -85,B 0,C 180,E1 20251.007,E2 20251.007} C_VEL
LIN {X 0,Y 511.91,Z 758.745,A -85,B 0,C 180,E1 20248.657,E2 20248.657} C_VEL
LIN {X 0,Y 511.914,Z 757.107,A -85,B 0,C 180,E1 20246.305,E2 20246.305} C_VEL
LIN {X 0,Y 511.936,Z 754.011,A -85,B 0,C 180,E1 20243.946,E2 20243.946} C_VEL
LIN {X 0,Y 511.983,Z 749.238,A -85,B 0,C 180,E1 20241.578,E2 20241.578} C_VEL
LIN {X 0,Y 512.11,Z 742.623,A -85,B 0,C 180,E1 20239.135,E2 20239.135} C_VEL
LIN {X 0,Y 512.355,Z 734.659,A -85,B 0,C 180,E1 20236.802,E2 20236.802} C_VEL
LIN {X 0,Y 512.727,Z 724.966,A -85,B 0,C 180,E1 20234.505,E2 20234.505} C_VEL
LIN {X 0,Y 513.291,Z 713.299,A -85,B 0,C 180,E1 20232.193,E2 20232.193} C_VEL
LIN {X 0,Y 514.045,Z 700.123,A -85,B 0,C 180,E1 20229.981,E2 20229.981} C_VEL
LIN {X 0,Y 514.939,Z 686.294,A -85,B 0,C 180,E1 20227.992,E2 20227.992} C_VEL
LIN {X 0,Y 515.982,Z 671.031,A -85,B 0,C 180,E1 20226.11,E2 20226.11} C_VEL
LIN {X 0,Y 517.262,Z 653.228,A -85,B 0,C 180,E1 20224.221,E2 20224.221} C_VEL
LIN {X 0,Y 518.537,Z 635.631,A -85,B 0,C 180,E1 20222.621,E2 20222.621} C_VEL
LIN {X 0,Y 519.853,Z 617.163,A -85,B 0,C 180,E1 20221.198,E2 20221.198} C_VEL
LIN {X 0,Y 521.141,Z 597.411,A -85,B 0,C 180,E1 20219.916,E2 20219.916} C_VEL
LIN {X 0,Y 522.409,Z 576.97,A -85,B 0,C 180,E1 20218.819,E2 20218.819} C_VEL
LIN {X 0,Y 523.437,Z 557.141,A -85,B 0,C 180,E1 20217.962,E2 20217.962} C_VEL
LIN {X 0,Y 524.339,Z 535.731,A -85,B 0,C 180,E1 20217.247,E2 20217.247} C_VEL
LIN {X 0,Y 525.064,Z 514.298,A -85,B 0,C 180,E1 20216.731,E2 20216.731} C_VEL
LIN {X 0,Y 528.126,Z 285.848,A -85,B 0,C 180,E1 20213.184,E2 20213.184} C_VEL
LIN {X 0,Y 528.914,Z 225.65,A -85,B 0,C 180,E1 20212.209,E2 20212.209} C_VEL
LIN {X 0,Y 525.912,Z 207.686,A -85,B 0,C 180,E1 20211.596,E2 20211.596} C_VEL
LIN {X 0,Y 527.877,Z 171.184,A -85,B 0,C 180,E1 20208.926,E2 20208.926} C_VEL
LIN {X 0,Y 520.621,Z 155.113,A -85,B 0,C 180,E1 20206.868,E2 20206.868} C_VEL
LIN {X 0,Y 514.256,Z 142.142,A -85,B 0,C 180,E1 20205.05,E2 20205.05} C_VEL
LIN {X 0,Y 512.652,Z 138.426,A -85,B 0,C 180,E1 20204.477,E2 20204.477} C_VEL
LIN {X 0,Y 512.585,Z 138.185,A -85,B 0,C 180,E1 20201.247,E2 20201.247} C_VEL
LIN {X 0,Y 512.568,Z 138.2,A -85,B 0,C 180,E1 20197.814,E2 20197.814} C_VEL
LIN {X 0,Y 512.61,Z 138.183,A -85,B 0,C 180,E1 20194.448,E2 20194.448} C_VEL
LIN {X 0,Y 512.586,Z 138.174,A -85,B 0,C 180,E1 20191.256,E2 20191.256} C_VEL
LIN {X 0,Y 512.58,Z 138.197,A -85,B 0,C 180,E1 20187.915,E2 20187.915} C_VEL
LIN {X 0,Y 512.628,Z 138.17,A -85,B 0,C 180,E1 20184.548,E2 20184.548} C_VEL
LIN {X 0,Y 512.598,Z 138.194,A -85,B 0,C 180,E1 20181.273,E2 20181.273} C_VEL
LIN {X 0,Y 512.588,Z 138.184,A -85,B 0,C 180,E1 20177.833,E2 20177.833} C_VEL
LIN {X 0,Y 512.631,Z 138.186,A -85,B 0,C 180,E1 20174.457,E2 20174.457} C_VEL
LIN {X 0,Y 512.629,Z 138.188,A -85,B 0,C 180,E1 20171.02,E2 20171.02} C_VEL
LIN {X 0,Y 512.595,Z 138.191,A -85,B 0,C 180,E1 20167.622,E2 20167.622} C_VEL
LIN {X 0,Y 512.612,Z 138.185,A -85,B 0,C 180,E1 20164.139,E2 20164.139} C_VEL
LIN {X 0,Y 512.652,Z 138.183,A -85,B 0,C 180,E1 20160.671,E2 20160.671} C_VEL
LIN {X 0,Y 512.624,Z 138.191,A -85,B 0,C 180,E1 20157.205,E2 20157.205} C_VEL
LIN {X 0,Y 512.608,Z 138.19,A -85,B 0,C 180,E1 20153.729,E2 20153.729} C_VEL
LIN {X 0,Y 512.637,Z 138.183,A -85,B 0,C 180,E1 20150.344,E2 20150.344} C_VEL
LIN {X 0,Y 512.646,Z 138.183,A -85,B 0,C 180,E1 20146.924,E2 20146.924} C_VEL
LIN {X 0,Y 512.619,Z 138.173,A -85,B 0,C 180,E1 20143.455,E2 20143.455} C_VEL
LIN {X 0,Y 512.621,Z 138.185,A -85,B 0,C 180,E1 20139.923,E2 20139.923} C_VEL
LIN {X 0,Y 512.649,Z 138.188,A -85,B 0,C 180,E1 20136.433,E2 20136.433} C_VEL
LIN {X 0,Y 512.641,Z 138.166,A -85,B 0,C 180,E1 20132.971,E2 20132.971} C_VEL
LIN {X 0,Y 512.629,Z 138.192,A -85,B 0,C 180,E1 20129.528,E2 20129.528} C_VEL
LIN {X 0,Y 512.632,Z 138.189,A -85,B 0,C 180,E1 20125.96,E2 20125.96} C_VEL
LIN {X 0,Y 512.641,Z 138.171,A -85,B 0,C 180,E1 20122.517,E2 20122.517} C_VEL
LIN {X 0,Y 512.64,Z 138.166,A -85,B 0,C 180,E1 20119.007,E2 20119.007} C_VEL
LIN {X 0,Y 512.673,Z 138.472,A -85,B 0,C 180,E1 20117.789,E2 20117.789} C_VEL
LIN {X 0,Y 514.204,Z 142.03,A -85,B 0,C 180,E1 20117.264,E2 20117.264} C_VEL
LIN {X 0,Y 521.362,Z 156.103,A -85,B 0,C 180,E1 20115.355,E2 20115.355} C_VEL
LIN {X 0,Y 525.191,Z 163.636,A -85,B 0,C 180,E1 20114.426,E2 20114.426} C_VEL
LIN {X 0,Y 532.633,Z 175.257,A -85,B 0,C 180,E1 20113.506,E2 20113.506} C_VEL
LIN {X 0,Y 533.799,Z 182.766,A -85,B 0,C 180,E1 20113.265,E2 20113.265} C_VEL
LIN {X 0,Y 531.289,Z 365.513,A -85,B 0,C 180,E1 20110.346,E2 20110.346} C_VEL
LIN {X 0,Y 529.053,Z 511.357,A -85,B 0,C 180,E1 20108.008,E2 20108.008} C_VEL
LIN {X 0,Y 528.199,Z 534.261,A -85,B 0,C 180,E1 20107.456,E2 20107.456} C_VEL
LIN {X 0,Y 527.201,Z 554.74,A -85,B 0,C 180,E1 20106.794,E2 20106.794} C_VEL
LIN {X 0,Y 525.863,Z 577.409,A -85,B 0,C 180,E1 20105.846,E2 20105.846} C_VEL
LIN {X 0,Y 524.538,Z 597.596,A -85,B 0,C 180,E1 20104.812,E2 20104.812} C_VEL
LIN {X 0,Y 522.891,Z 619.151,A -85,B 0,C 180,E1 20103.48,E2 20103.48} C_VEL
LIN {X 0,Y 521.357,Z 638.981,A -85,B 0,C 180,E1 20102.041,E2 20102.041} C_VEL
LIN {X 0,Y 519.728,Z 658.279,A -85,B 0,C 180,E1 20100.394,E2 20100.394} C_VEL
LIN {X 0,Y 518.081,Z 678.141,A -85,B 0,C 180,E1 20098.429,E2 20098.429} C_VEL
LIN {X 0,Y 516.735,Z 694.666,A -85,B 0,C 180,E1 20096.549,E2 20096.549} C_VEL
LIN {X 0,Y 515.53,Z 710.15,A -85,B 0,C 180,E1 20094.522,E2 20094.522} C_VEL
LIN {X 0,Y 514.471,Z 725.224,A -85,B 0,C 180,E1 20092.27,E2 20092.27} C_VEL
LIN {X 0,Y 513.634,Z 738.093,A -85,B 0,C 180,E1 20090.035,E2 20090.035} C_VEL
LIN {X 0,Y 512.97,Z 750.287,A -85,B 0,C 180,E1 20087.584,E2 20087.584} C_VEL
LIN {X 0,Y 512.526,Z 760.072,A -85,B 0,C 180,E1 20085.269,E2 20085.269} C_VEL
LIN {X 0,Y 512.212,Z 768.991,A -85,B 0,C 180,E1 20082.743,E2 20082.743} C_VEL
LIN {X 0,Y 512.06,Z 775.564,A -85,B 0,C 180,E1 20080.462,E2 20080.462} C_VEL
LIN {X 0,Y 511.965,Z 781.428,A -85,B 0,C 180,E1 20077.857,E2 20077.857} C_VEL
LIN {X 0,Y 511.911,Z 785.118,A -85,B 0,C 180,E1 20075.604,E2 20075.604} C_VEL
LIN {X 0,Y 511.913,Z 787.851,A -85,B 0,C 180,E1 20073.023,E2 20073.023} C_VEL
LIN {X 0,Y 511.9,Z 788.872,A -85,B 0,C 180,E1 20070.671,E2 20070.671} C_VEL
LIN {X 0,Y 511.906,Z 788.526,A -85,B 0,C 180,E1 20068.097,E2 20068.097} C_VEL
LIN {X 0,Y 511.905,Z 786.729,A -85,B 0,C 180,E1 20065.744,E2 20065.744} C_VEL
LIN {X 0,Y 511.941,Z 783.494,A -85,B 0,C 180,E1 20063.271,E2 20063.271} C_VEL
LIN {X 0,Y 512,Z 778.574,A -85,B 0,C 180,E1 20060.786,E2 20060.786} C_VEL
LIN {X 0,Y 512.141,Z 772.176,A -85,B 0,C 180,E1 20058.286,E2 20058.286} C_VEL
LIN {X 0,Y 512.366,Z 764.344,A -85,B 0,C 180,E1 20055.882,E2 20055.882} C_VEL
LIN {X 0,Y 512.779,Z 754.425,A -85,B 0,C 180,E1 20053.344,E2 20053.344} C_VEL
LIN {X 0,Y 513.326,Z 743.575,A -85,B 0,C 180,E1 20051.018,E2 20051.018} C_VEL
LIN {X 0,Y 514.125,Z 730.162,A -85,B 0,C 180,E1 20048.555,E2 20048.555} C_VEL
LIN {X 0,Y 515.118,Z 716.014,A -85,B 0,C 180,E1 20046.31,E2 20046.31} C_VEL
LIN {X 0,Y 516.284,Z 700.343,A -85,B 0,C 180,E1 20044.168,E2 20044.168} C_VEL
LIN {X 0,Y 517.696,Z 682.786,A -85,B 0,C 180,E1 20042.073,E2 20042.073} C_VEL
LIN {X 0,Y 519.121,Z 665.69,A -85,B 0,C 180,E1 20040.302,E2 20040.302} C_VEL
LIN {X 0,Y 520.754,Z 645.803,A -85,B 0,C 180,E1 20038.518,E2 20038.518} C_VEL
LIN {X 0,Y 522.439,Z 625.552,A -85,B 0,C 180,E1 20036.956,E2 20036.956} C_VEL
LIN {X 0,Y 523.97,Z 604.835,A -85,B 0,C 180,E1 20035.61,E2 20035.61} C_VEL
LIN {X 0,Y 525.562,Z 582.547,A -85,B 0,C 180,E1 20034.399,E2 20034.399} C_VEL
LIN {X 0,Y 526.757,Z 562.739,A -85,B 0,C 180,E1 20033.518,E2 20033.518} C_VEL
LIN {X 0,Y 527.946,Z 539.524,A -85,B 0,C 180,E1 20032.695,E2 20032.695} C_VEL
LIN {X 0,Y 528.804,Z 518.591,A -85,B 0,C 180,E1 20032.145,E2 20032.145} C_VEL
LIN {X 0,Y 529.501,Z 487.99,A -85,B 0,C 180,E1 20031.597,E2 20031.597} C_VEL
LIN {X 0,Y 532.528,Z 280.037,A -85,B 0,C 180,E1 20028.287,E2 20028.287} C_VEL
LIN {X 0,Y 533.665,Z 180.885,A -85,B 0,C 180,E1 20026.689,E2 20026.689} C_VEL
LIN {X 0,Y 532.321,Z 174.482,A -85,B 0,C 180,E1 20026.451,E2 20026.451} C_VEL
LIN {X 0,Y 524.39,Z 162.353,A -85,B 0,C 180,E1 20025.441,E2 20025.441} C_VEL
LIN {X 0,Y 516.675,Z 146.677,A -85,B 0,C 180,E1 20023.392,E2 20023.392} C_VEL
LIN {X 0,Y 514.204,Z 142.03,A -85,B 0,C 180,E1 20022.736,E2 20022.736} C_VEL
LIN {X 0,Y 512.675,Z 138.475,A -85,B 0,C 180,E1 20022.211,E2 20022.211} C_VEL
LIN {X 0,Y 512.633,Z 138.168,A -85,B 0,C 180,E1 20020.479,E2 20020.479} C_VEL
LIN {X 0,Y 512.639,Z 138.168,A -85,B 0,C 180,E1 20017.062,E2 20017.062} C_VEL
LIN {X 0,Y 512.642,Z 138.178,A -85,B 0,C 180,E1 20013.502,E2 20013.502} C_VEL
LIN {X 0,Y 512.632,Z 138.191,A -85,B 0,C 180,E1 20010.006,E2 20010.006} C_VEL
LIN {X 0,Y 512.625,Z 138.173,A -85,B 0,C 180,E1 20006.461,E2 20006.461} C_VEL
LIN {X 0,Y 512.648,Z 138.174,A -85,B 0,C 180,E1 20002.959,E2 20002.959} C_VEL
LIN {X 0,Y 512.647,Z 138.184,A -85,B 0,C 180,E1 19999.364,E2 19999.364} C_VEL
LIN {X 0,Y 512.623,Z 138.166,A -85,B 0,C 180,E1 19995.939,E2 19995.939} C_VEL
LIN {X 0,Y 512.615,Z 138.192,A -85,B 0,C 180,E1 19992.389,E2 19992.389} C_VEL
LIN {X 0,Y 512.64,Z 138.193,A -85,B 0,C 180,E1 19988.863,E2 19988.863} C_VEL
LIN {X 0,Y 512.648,Z 138.188,A -85,B 0,C 180,E1 19985.372,E2 19985.372} C_VEL
LIN {X 0,Y 512.618,Z 138.19,A -85,B 0,C 180,E1 19981.9,E2 19981.9} C_VEL
LIN {X 0,Y 512.607,Z 138.194,A -85,B 0,C 180,E1 19978.435,E2 19978.435} C_VEL
LIN {X 0,Y 512.643,Z 138.189,A -85,B 0,C 180,E1 19975.077,E2 19975.077} C_VEL
LIN {X 0,Y 512.62,Z 138.188,A -85,B 0,C 180,E1 19971.701,E2 19971.701} C_VEL
LIN {X 0,Y 512.596,Z 138.193,A -85,B 0,C 180,E1 19968.283,E2 19968.283} C_VEL
LIN {X 0,Y 512.62,Z 138.193,A -85,B 0,C 180,E1 19964.849,E2 19964.849} C_VEL
LIN {X 0,Y 512.639,Z 138.166,A -85,B 0,C 180,E1 19961.419,E2 19961.419} C_VEL
LIN {X 0,Y 512.593,Z 138.194,A -85,B 0,C 180,E1 19958.006,E2 19958.006} C_VEL
LIN {X 0,Y 512.586,Z 138.17,A -85,B 0,C 180,E1 19954.463,E2 19954.463} C_VEL
LIN {X 0,Y 512.632,Z 138.188,A -85,B 0,C 180,E1 19951.072,E2 19951.072} C_VEL
LIN {X 0,Y 512.592,Z 138.185,A -85,B 0,C 180,E1 19947.825,E2 19947.825} C_VEL
LIN {X 0,Y 512.575,Z 138.172,A -85,B 0,C 180,E1 19944.43,E2 19944.43} C_VEL
LIN {X 0,Y 512.625,Z 138.183,A -85,B 0,C 180,E1 19941.093,E2 19941.093} C_VEL
LIN {X 0,Y 512.592,Z 138.199,A -85,B 0,C 180,E1 19937.704,E2 19937.704} C_VEL
LIN {X 0,Y 512.622,Z 138.276,A -85,B 0,C 180,E1 19935.485,E2 19935.485} C_VEL
LIN {X 0,Y 512.706,Z 138.697,A -85,B 0,C 180,E1 19935.366,E2 19935.366} C_VEL
LIN {X 0,Y 514.502,Z 143.486,A -85,B 0,C 180,E1 19934.714,E2 19934.714} C_VEL
LIN {X 0,Y 515.183,Z 151.074,A -85,B 0,C 180,E1 19933.98,E2 19933.98} C_VEL
LIN {X 0,Y 515.887,Z 161.455,A -85,B 0,C 180,E1 19933.025,E2 19933.025} C_VEL
LIN {X 0,Y 516.742,Z 164.473,A -85,B 0,C 180,E1 19932.673,E2 19932.673} C_VEL
LIN {X 0,Y 521.404,Z 175.278,A -85,B 0,C 180,E1 19931.299,E2 19931.299} C_VEL
LIN {X 0,Y 519.521,Z 208.065,A -85,B 0,C 180,E1 19928.899,E2 19928.899} C_VEL
LIN {X 0,Y 522.958,Z 229.264,A -85,B 0,C 180,E1 19928.196,E2 19928.196} C_VEL
LIN {X 0,Y 519.184,Z 461.114,A -85,B 0,C 180,E1 19924.509,E2 19924.509} C_VEL
LIN {X 0,Y 518.325,Z 516.468,A -85,B 0,C 180,E1 19923.624,E2 19923.624} C_VEL
LIN {X 0,Y 517.502,Z 537.715,A -85,B 0,C 180,E1 19923.087,E2 19923.087} C_VEL
LIN {X 0,Y 516.477,Z 559.462,A -85,B 0,C 180,E1 19922.329,E2 19922.329} C_VEL
LIN {X 0,Y 515.319,Z 579.731,A -85,B 0,C 180,E1 19921.425,E2 19921.425} C_VEL
LIN {X 0,Y 513.936,Z 600.006,A -85,B 0,C 180,E1 19920.293,E2 19920.293} C_VEL
LIN {X 0,Y 512.462,Z 620.067,A -85,B 0,C 180,E1 19918.938,E2 19918.938} C_VEL
LIN {X 0,Y 511.07,Z 638.127,A -85,B 0,C 180,E1 19917.497,E2 19917.497} C_VEL
LIN {X 0,Y 509.637,Z 655.984,A -85,B 0,C 180,E1 19915.819,E2 19915.819} C_VEL
LIN {X 0,Y 508.344,Z 672.311,A -85,B 0,C 180,E1 19914.025,E2 19914.025} C_VEL
LIN {X 0,Y 507.146,Z 688.216,A -85,B 0,C 180,E1 19911.998,E2 19911.998} C_VEL
LIN {X 0,Y 506.169,Z 702.335,A -85,B 0,C 180,E1 19909.904,E2 19909.904} C_VEL
LIN {X 0,Y 505.378,Z 714.718,A -85,B 0,C 180,E1 19907.738,E2 19907.738} C_VEL
LIN {X 0,Y 504.768,Z 726.121,A -85,B 0,C 180,E1 19905.392,E2 19905.392} C_VEL
LIN {X 0,Y 504.37,Z 735.601,A -85,B 0,C 180,E1 19903.061,E2 19903.061} C_VEL
LIN {X 0,Y 504.122,Z 743.245,A -85,B 0,C 180,E1 19900.745,E2 19900.745} C_VEL
LIN {X 0,Y 503.993,Z 749.547,A -85,B 0,C 180,E1 19898.327,E2 19898.327} C_VEL
LIN {X 0,Y 503.937,Z 754.254,A -85,B 0,C 180,E1 19895.922,E2 19895.922} C_VEL
LIN {X 0,Y 503.913,Z 757.242,A -85,B 0,C 180,E1 19893.526,E2 19893.526} C_VEL
LIN {X 0,Y 503.912,Z 758.793,A -85,B 0,C 180,E1 19891.023,E2 19891.023} C_VEL
LIN {X 0,Y 503.91,Z 758.745,A -85,B 0,C 180,E1 19888.636,E2 19888.636} C_VEL
LIN {X 0,Y 503.914,Z 757.106,A -85,B 0,C 180,E1 19886.246,E2 19886.246} C_VEL
LIN {X 0,Y 503.938,Z 754.01,A -85,B 0,C 180,E1 19883.85,E2 19883.85} C_VEL
LIN {X 0,Y 503.989,Z 749.237,A -85,B 0,C 180,E1 19881.443,E2 19881.443} C_VEL
LIN {X 0,Y 504.133,Z 742.813,A -85,B 0,C 180,E1 19879.024,E2 19879.024} C_VEL
LIN {X 0,Y 504.397,Z 735.099,A -85,B 0,C 180,E1 19876.707,E2 19876.707} C_VEL
LIN {X 0,Y 504.807,Z 725.483,A -85,B 0,C 180,E1 19874.374,E2 19874.374} C_VEL
LIN {X 0,Y 505.425,Z 713.929,A -85,B 0,C 180,E1 19872.025,E2 19872.025} C_VEL
LIN {X 0,Y 506.208,Z 701.659,A -85,B 0,C 180,E1 19869.899,E2 19869.899} C_VEL
LIN {X 0,Y 507.221,Z 687.14,A -85,B 0,C 180,E1 19867.761,E2 19867.761} C_VEL
LIN {X 0,Y 508.404,Z 671.532,A -85,B 0,C 180,E1 19865.793,E2 19865.793} C_VEL
LIN {X 0,Y 509.764,Z 654.437,A -85,B 0,C 180,E1 19863.938,E2 19863.938} C_VEL
LIN {X 0,Y 511.202,Z 636.352,A -85,B 0,C 180,E1 19862.258,E2 19862.258} C_VEL
LIN {X 0,Y 512.632,Z 617.963,A -85,B 0,C 180,E1 19860.817,E2 19860.817} C_VEL
LIN {X 0,Y 514.066,Z 597.955,A -85,B 0,C 180,E1 19859.494,E2 19859.494} C_VEL
LIN {X 0,Y 515.454,Z 577.582,A -85,B 0,C 180,E1 19858.382,E2 19858.382} C_VEL
LIN {X 0,Y 516.605,Z 557.046,A -85,B 0,C 180,E1 19857.483,E2 19857.483} C_VEL
LIN {X 0,Y 517.589,Z 535.789,A -85,B 0,C 180,E1 19856.768,E2 19856.768} C_VEL
LIN {X 0,Y 518.365,Z 514.641,A -85,B 0,C 180,E1 19856.251,E2 19856.251} C_VEL
LIN {X 0,Y 522.076,Z 280.714,A -85,B 0,C 180,E1 19852.537,E2 19852.537} C_VEL
LIN {X 0,Y 522.811,Z 227.224,A -85,B 0,C 180,E1 19851.665,E2 19851.665} C_VEL
LIN {X 0,Y 519.459,Z 207.061,A -85,B 0,C 180,E1 19850.959,E2 19850.959} C_VEL
LIN {X 0,Y 521.342,Z 174.906,A -85,B 0,C 180,E1 19848.575,E2 19848.575} C_VEL
LIN {X 0,Y 514.562,Z 159.872,A -85,B 0,C 180,E1 19846.613,E2 19846.613} C_VEL
LIN {X 0,Y 506.3,Z 143.125,A -85,B 0,C 180,E1 19844.196,E2 19844.196} C_VEL
LIN {X 0,Y 504.696,Z 139.582,A -85,B 0,C 180,E1 19843.644,E2 19843.644} C_VEL
LIN {X 0,Y 504.657,Z 139.165,A -85,B 0,C 180,E1 19843.121,E2 19843.121} C_VEL
LIN {X 0,Y 504.627,Z 139.164,A -85,B 0,C 180,E1 19839.758,E2 19839.758} C_VEL
LIN {X 0,Y 504.668,Z 139.158,A -85,B 0,C 180,E1 19836.452,E2 19836.452} C_VEL
LIN {X 0,Y 504.671,Z 139.186,A -85,B 0,C 180,E1 19833.013,E2 19833.013} C_VEL
LIN {X 0,Y 504.635,Z 139.174,A -85,B 0,C 180,E1 19829.692,E2 19829.692} C_VEL
LIN {X 0,Y 504.668,Z 139.163,A -85,B 0,C 180,E1 19826.346,E2 19826.346} C_VEL
LIN {X 0,Y 504.698,Z 139.179,A -85,B 0,C 180,E1 19822.849,E2 19822.849} C_VEL
LIN {X 0,Y 504.65,Z 139.155,A -85,B 0,C 180,E1 19819.427,E2 19819.427} C_VEL
LIN {X 0,Y 504.651,Z 139.184,A -85,B 0,C 180,E1 19815.868,E2 19815.868} C_VEL
LIN {X 0,Y 504.694,Z 139.18,A -85,B 0,C 180,E1 19812.471,E2 19812.471} C_VEL
LIN {X 0,Y 504.695,Z 139.184,A -85,B 0,C 180,E1 19809.004,E2 19809.004} C_VEL
LIN {X 0,Y 504.659,Z 139.183,A -85,B 0,C 180,E1 19805.685,E2 19805.685} C_VEL
LIN {X 0,Y 504.676,Z 139.181,A -85,B 0,C 180,E1 19802.157,E2 19802.157} C_VEL
LIN {X 0,Y 504.712,Z 139.181,A -85,B 0,C 180,E1 19798.752,E2 19798.752} C_VEL
LIN {X 0,Y 504.686,Z 139.181,A -85,B 0,C 180,E1 19795.227,E2 19795.227} C_VEL
LIN {X 0,Y 504.671,Z 139.179,A -85,B 0,C 180,E1 19791.799,E2 19791.799} C_VEL
LIN {X 0,Y 504.699,Z 139.177,A -85,B 0,C 180,E1 19788.342,E2 19788.342} C_VEL
LIN {X 0,Y 504.707,Z 139.146,A -85,B 0,C 180,E1 19784.841,E2 19784.841} C_VEL
LIN {X 0,Y 504.695,Z 139.183,A -85,B 0,C 180,E1 19781.28,E2 19781.28} C_VEL
LIN {X 0,Y 504.679,Z 139.154,A -85,B 0,C 180,E1 19777.765,E2 19777.765} C_VEL
LIN {X 0,Y 504.703,Z 139.171,A -85,B 0,C 180,E1 19774.288,E2 19774.288} C_VEL
LIN {X 0,Y 504.705,Z 139.179,A -85,B 0,C 180,E1 19770.704,E2 19770.704} C_VEL
LIN {X 0,Y 504.704,Z 139.155,A -85,B 0,C 180,E1 19767.125,E2 19767.125} C_VEL
LIN {X 0,Y 504.689,Z 139.158,A -85,B 0,C 180,E1 19763.676,E2 19763.676} C_VEL
LIN {X 0,Y 504.707,Z 139.163,A -85,B 0,C 180,E1 19760.217,E2 19760.217} C_VEL
LIN {X 0,Y 504.713,Z 139.274,A -85,B 0,C 180,E1 19758.724,E2 19758.724} C_VEL
LIN {X 0,Y 505.136,Z 140.94,A -85,B 0,C 180,E1 19758.433,E2 19758.433} C_VEL
LIN {X 0,Y 507.366,Z 145.113,A -85,B 0,C 180,E1 19757.813,E2 19757.813} C_VEL
LIN {X 0,Y 513.936,Z 158.003,A -85,B 0,C 180,E1 19756.01,E2 19756.01} C_VEL
LIN {X 0,Y 517.164,Z 164.257,A -85,B 0,C 180,E1 19755.214,E2 19755.214} C_VEL
LIN {X 0,Y 526.999,Z 179.359,A -85,B 0,C 180,E1 19753.964,E2 19753.964} C_VEL
LIN {X 0,Y 527.699,Z 184.682,A -85,B 0,C 180,E1 19753.801,E2 19753.801} C_VEL
LIN {X 0,Y 524.779,Z 390.148,A -85,B 0,C 180,E1 19750.513,E2 19750.513} C_VEL
LIN {X 0,Y 522.745,Z 511.357,A -85,B 0,C 180,E1 19748.55,E2 19748.55} C_VEL
LIN {X 0,Y 521.832,Z 534.129,A -85,B 0,C 180,E1 19747.998,E2 19747.998} C_VEL
LIN {X 0,Y 520.797,Z 553.887,A -85,B 0,C 180,E1 19747.356,E2 19747.356} C_VEL
LIN {X 0,Y 519.341,Z 576.527,A -85,B 0,C 180,E1 19746.414,E2 19746.414} C_VEL
LIN {X 0,Y 517.914,Z 596.476,A -85,B 0,C 180,E1 19745.391,E2 19745.391} C_VEL
LIN {X 0,Y 516.14,Z 618.248,A -85,B 0,C 180,E1 19744.044,E2 19744.044} C_VEL
LIN {X 0,Y 514.406,Z 638.43,A -85,B 0,C 180,E1 19742.574,E2 19742.574} C_VEL
LIN {X 0,Y 512.672,Z 657.422,A -85,B 0,C 180,E1 19740.941,E2 19740.941} C_VEL
LIN {X 0,Y 510.957,Z 676.129,A -85,B 0,C 180,E1 19739.095,E2 19739.095} C_VEL
LIN {X 0,Y 509.467,Z 692.638,A -85,B 0,C 180,E1 19737.211,E2 19737.211} C_VEL
LIN {X 0,Y 508.031,Z 709.303,A -85,B 0,C 180,E1 19735.032,E2 19735.032} C_VEL
LIN {X 0,Y 506.835,Z 724.511,A -85,B 0,C 180,E1 19732.746,E2 19732.746} C_VEL
LIN {X 0,Y 505.852,Z 738.091,A -85,B 0,C 180,E1 19730.357,E2 19730.357} C_VEL
LIN {X 0,Y 505.09,Z 750.617,A -85,B 0,C 180,E1 19727.793,E2 19727.793} C_VEL
LIN {X 0,Y 504.609,Z 760.071,A -85,B 0,C 180,E1 19725.515,E2 19725.515} C_VEL
LIN {X 0,Y 504.241,Z 769.348,A -85,B 0,C 180,E1 19722.831,E2 19722.831} C_VEL
LIN {X 0,Y 504.072,Z 775.867,A -85,B 0,C 180,E1 19720.514,E2 19720.514} C_VEL
LIN {X 0,Y 503.968,Z 781.635,A -85,B 0,C 180,E1 19717.868,E2 19717.868} C_VEL
LIN {X 0,Y 503.912,Z 785.278,A -85,B 0,C 180,E1 19715.579,E2 19715.579} C_VEL
LIN {X 0,Y 503.914,Z 787.919,A -85,B 0,C 180,E1 19712.957,E2 19712.957} C_VEL
LIN {X 0,Y 503.9,Z 788.872,A -85,B 0,C 180,E1 19710.682,E2 19710.682} C_VEL
LIN {X 0,Y 503.907,Z 788.526,A -85,B 0,C 180,E1 19708.067,E2 19708.067} C_VEL
LIN {X 0,Y 503.904,Z 786.729,A -85,B 0,C 180,E1 19705.676,E2 19705.676} C_VEL
LIN {X 0,Y 503.944,Z 783.494,A -85,B 0,C 180,E1 19703.163,E2 19703.163} C_VEL
LIN {X 0,Y 504.007,Z 778.574,A -85,B 0,C 180,E1 19700.638,E2 19700.638} C_VEL
LIN {X 0,Y 504.169,Z 772.175,A -85,B 0,C 180,E1 19698.098,E2 19698.098} C_VEL
LIN {X 0,Y 504.428,Z 764.345,A -85,B 0,C 180,E1 19695.655,E2 19695.655} C_VEL
LIN {X 0,Y 504.893,Z 754.424,A -85,B 0,C 180,E1 19693.076,E2 19693.076} C_VEL
LIN {X 0,Y 505.506,Z 743.577,A -85,B 0,C 180,E1 19690.713,E2 19690.713} C_VEL
LIN {X 0,Y 506.401,Z 730.16,A -85,B 0,C 180,E1 19688.211,E2 19688.211} C_VEL
LIN {X 0,Y 507.495,Z 716.016,A -85,B 0,C 180,E1 19685.932,E2 19685.932} C_VEL
LIN {X 0,Y 508.793,Z 700.342,A -85,B 0,C 180,E1 19683.759,E2 19683.759} C_VEL
LIN {X 0,Y 510.309,Z 683.339,A -85,B 0,C 180,E1 19681.697,E2 19681.697} C_VEL
LIN {X 0,Y 511.832,Z 666.552,A -85,B 0,C 180,E1 19679.928,E2 19679.928} C_VEL
LIN {X 0,Y 513.654,Z 646.533,A -85,B 0,C 180,E1 19678.097,E2 19678.097} C_VEL
LIN {X 0,Y 515.412,Z 627.098,A -85,B 0,C 180,E1 19676.57,E2 19676.57} C_VEL
LIN {X 0,Y 517.065,Z 606.841,A -85,B 0,C 180,E1 19675.22,E2 19675.22} C_VEL
LIN {X 0,Y 518.716,Z 586.199,A -85,B 0,C 180,E1 19674.054,E2 19674.054} C_VEL
LIN {X 0,Y 520.147,Z 564.548,A -85,B 0,C 180,E1 19673.062,E2 19673.062} C_VEL
LIN {X 0,Y 521.414,Z 542.767,A -85,B 0,C 180,E1 19672.254,E2 19672.254} C_VEL
LIN {X 0,Y 522.394,Z 520.539,A -85,B 0,C 180,E1 19671.649,E2 19671.649} C_VEL
LIN {X 0,Y 523.126,Z 495.164,A -85,B 0,C 180,E1 19671.166,E2 19671.166} C_VEL
LIN {X 0,Y 525.547,Z 330.211,A -85,B 0,C 180,E1 19668.541,E2 19668.541} C_VEL
LIN {X 0,Y 527.602,Z 182.695,A -85,B 0,C 180,E1 19666.154,E2 19666.154} C_VEL
LIN {X 0,Y 526.617,Z 178.552,A -85,B 0,C 180,E1 19665.985,E2 19665.985} C_VEL
LIN {X 0,Y 516.409,Z 163.042,A -85,B 0,C 180,E1 19664.654,E2 19664.654} C_VEL
LIN {X 0,Y 508.674,Z 147.569,A -85,B 0,C 180,E1 19662.545,E2 19662.545} C_VEL
LIN {X 0,Y 506.259,Z 143.003,A -85,B 0,C 180,E1 19661.878,E2 19661.878} C_VEL
LIN {X 0,Y 504.746,Z 139.488,A -85,B 0,C 180,E1 19661.345,E2 19661.345} C_VEL
LIN {X 0,Y 504.692,Z 139.156,A -85,B 0,C 180,E1 19660.378,E2 19660.378} C_VEL
LIN {X 0,Y 504.702,Z 139.154,A -85,B 0,C 180,E1 19656.889,E2 19656.889} C_VEL
LIN {X 0,Y 504.702,Z 139.163,A -85,B 0,C 180,E1 19653.418,E2 19653.418} C_VEL
LIN {X 0,Y 504.695,Z 139.18,A -85,B 0,C 180,E1 19649.95,E2 19649.95} C_VEL
LIN {X 0,Y 504.686,Z 139.16,A -85,B 0,C 180,E1 19646.433,E2 19646.433} C_VEL
LIN {X 0,Y 504.707,Z 139.161,A -85,B 0,C 180,E1 19642.902,E2 19642.902} C_VEL
LIN {X 0,Y 504.708,Z 139.173,A -85,B 0,C 180,E1 19639.319,E2 19639.319} C_VEL
LIN {X 0,Y 504.687,Z 139.151,A -85,B 0,C 180,E1 19635.866,E2 19635.866} C_VEL
LIN {X 0,Y 504.677,Z 139.181,A -85,B 0,C 180,E1 19632.355,E2 19632.355} C_VEL
LIN {X 0,Y 504.702,Z 139.181,A -85,B 0,C 180,E1 19628.889,E2 19628.889} C_VEL
LIN {X 0,Y 504.71,Z 139.177,A -85,B 0,C 180,E1 19625.342,E2 19625.342} C_VEL
LIN {X 0,Y 504.684,Z 139.179,A -85,B 0,C 180,E1 19621.816,E2 19621.816} C_VEL
LIN {X 0,Y 504.667,Z 139.182,A -85,B 0,C 180,E1 19618.297,E2 19618.297} C_VEL
LIN {X 0,Y 504.692,Z 139.183,A -85,B 0,C 180,E1 19614.885,E2 19614.885} C_VEL
LIN {X 0,Y 504.704,Z 139.176,A -85,B 0,C 180,E1 19611.455,E2 19611.455} C_VEL
LIN {X 0,Y 504.662,Z 139.181,A -85,B 0,C 180,E1 19607.993,E2 19607.993} C_VEL
LIN {X 0,Y 504.659,Z 139.184,A -85,B 0,C 180,E1 19604.486,E2 19604.486} C_VEL
